LIN {X 0,Y 210.828,Z 695.055,A -85,B 0,C 180,E1 -21900.557,E2 -21900.557} C_VEL
LIN {X 0,Y 214.212,Z 683.602,A -85,B 0,C 180,E1 -21902.499,E2 -21902.499} C_VEL
LIN {X 0,Y 216.871,Z 672.44,A -85,B 0,C 180,E1 -21903.99,E2 -21903.99} C_VEL
LIN {X 0,Y 219.279,Z 660.117,A -85,B 0,C 180,E1 -21905.236,E2 -21905.236} C_VEL
LIN {X 0,Y 220.903,Z 648.24,A -85,B 0,C 180,E1 -21906.129,E2 -21906.129} C_VEL
LIN {X 0,Y 222.158,Z 635.708,A -85,B 0,C 180,E1 -21906.737,E2 -21906.737} C_VEL
LIN {X 0,Y 225.382,Z 570.119,A -85,B 0,C 180,E1 -21908.634,E2 -21908.634} C_VEL
LIN {X 0,Y 224.372,Z 564.639,A -85,B 0,C 180,E1 -21909.068,E2 -21909.068} C_VEL
LIN {X 0,Y 218.505,Z 551.425,A -85,B 0,C 180,E1 -21910.952,E2 -21910.952} C_VEL
LIN {X 0,Y 212.899,Z 540.525,A -85,B 0,C 180,E1 -21912.833,E2 -21912.833} C_VEL
LIN {X 0,Y 207.547,Z 531.361,A -85,B 0,C 180,E1 -21914.735,E2 -21914.735} C_VEL
LIN {X 0,Y 204.869,Z 527.036,A -85,B 0,C 180,E1 -21915.738,E2 -21915.738} C_VEL
LIN {X 0,Y 202.022,Z 522.55,A -85,B 0,C 180,E1 -21916.851,E2 -21916.851} C_VEL
LIN {X 0,Y 199.415,Z 518.27,A -85,B 0,C 180,E1 -21917.962,E2 -21917.962} C_VEL
LIN {X 0,Y 197.926,Z 513.312,A -85,B 0,C 180,E1 -21921.372,E2 -21921.372} C_VEL
LIN {X 0,Y 197,Z 511.784,A -85,B 0,C 180,E1 -21922.664,E2 -21922.664} C_VEL
LIN {X 0,Y 195.61,Z 510.693,A -85,B 0,C 180,E1 -21924.04,E2 -21924.04} C_VEL
LIN {X 0,Y 199.723,Z 529.401,A -85,B 0,C 180,E1 -21929.32,E2 -21929.32} C_VEL
LIN {X 0,Y 199.82,Z 531.676,A -85,B 0,C 180,E1 -21929.92,E2 -21929.92} C_VEL
LIN {X 0,Y 199.088,Z 537.434,A -85,B 0,C 180,E1 -21931.377,E2 -21931.377} C_VEL
LIN {X 0,Y 200.579,Z 559.049,A -85,B 0,C 180,E1 -21932.803,E2 -21932.803} C_VEL
LIN {X 0,Y 201.371,Z 568.64,A -85,B 0,C 180,E1 -21933.438,E2 -21933.438} C_VEL
LIN {X 0,Y 197.17,Z 649.531,A -85,B 0,C 180,E1 -21938.537,E2 -21938.537} C_VEL
LIN {X 0,Y 196.297,Z 664.074,A -85,B 0,C 180,E1 -21939.842,E2 -21939.842} C_VEL
LIN {X 0,Y 195.289,Z 676.673,A -85,B 0,C 180,E1 -21941.374,E2 -21941.374} C_VEL
LIN {X 0,Y 194.349,Z 688.461,A -85,B 0,C 180,E1 -21943.184,E2 -21943.184} C_VEL
LIN {X 0,Y 193.196,Z 700.417,A -85,B 0,C 180,E1 -21945.516,E2 -21945.516} C_VEL
LIN {X 0,Y 192.294,Z 710.299,A -85,B 0,C 180,E1 -21947.868,E2 -21947.868} C_VEL
LIN {X 0,Y 191.618,Z 719.434,A -85,B 0,C 180,E1 -21950.5,E2 -21950.5} C_VEL
LIN {X 0,Y 190.999,Z 728.454,A -85,B 0,C 180,E1 -21953.662,E2 -21953.662} C_VEL
LIN {X 0,Y 190.744,Z 735.772,A -85,B 0,C 180,E1 -21956.831,E2 -21956.831} C_VEL
LIN {X 0,Y 190.589,Z 741.573,A -85,B 0,C 180,E1 -21960,E2 -21960} C_VEL
LIN {X 0,Y 190.77,Z 746.231,A -85,B 0,C 180,E1 -21963.167,E2 -21963.167} C_VEL
LIN {X 0,Y 191.186,Z 749.856,A -85,B 0,C 180,E1 -21966.331,E2 -21966.331} C_VEL
LIN {X 0,Y 192.742,Z 753.216,A -85,B 0,C 180,E1 -21970.504,E2 -21970.504} C_VEL
LIN {X 0,Y 195.223,Z 755.083,A -85,B 0,C 180,E1 -21974.596,E2 -21974.596} C_VEL
LIN {X 0,Y 198.727,Z 755.426,A -85,B 0,C 180,E1 -21978.559,E2 -21978.559} C_VEL
LIN {X 0,Y 200.496,Z 755.13,A -85,B 0,C 180,E1 -21980.073,E2 -21980.073} C_VEL
LIN {X 0,Y 201.902,Z 754.816,A -85,B 0,C 180,E1 -21981.708,E2 -21981.708} C_VEL
LIN {X 0,Y 202.92,Z 754.106,A -85,B 0,C 180,E1 -21984.496,E2 -21984.496} C_VEL
LIN {X 0,Y 204.459,Z 752.722,A -85,B 0,C 180,E1 -21987.21,E2 -21987.21} C_VEL
LIN {X 0,Y 206.611,Z 751.36,A -85,B 0,C 180,E1 -21988.685,E2 -21988.685} C_VEL
LIN {X 0,Y 211.655,Z 748.402,A -85,B 0,C 180,E1 -21990.976,E2 -21990.976} C_VEL
LIN {X 0,Y 217.634,Z 744.305,A -85,B 0,C 180,E1 -21993.297,E2 -21993.297} C_VEL
LIN {X 0,Y 226.261,Z 737.268,A -85,B 0,C 180,E1 -21996.169,E2 -21996.169} C_VEL
LIN {X 0,Y 234.4,Z 729.413,A -85,B 0,C 180,E1 -21998.473,E2 -21998.473} C_VEL
LIN {X 0,Y 241.755,Z 721.254,A -85,B 0,C 180,E1 -22000.296,E2 -22000.296} C_VEL
LIN {X 0,Y 249.501,Z 711.354,A -85,B 0,C 180,E1 -22001.989,E2 -22001.989} C_VEL
LIN {X 0,Y 256.259,Z 701.388,A -85,B 0,C 180,E1 -22003.285,E2 -22003.285} C_VEL
LIN {X 0,Y 257.647,Z 699.121,A -85,B 0,C 180,E1 -22003.543,E2 -22003.543} C_VEL
LIN {X 0,Y 256.765,Z 700.563,A -85,B 0,C 180,E1 -22004.067,E2 -22004.067} C_VEL
LIN {X 0,Y 249.452,Z 711.541,A -85,B 0,C 180,E1 -22005.221,E2 -22005.221} C_VEL
LIN {X 0,Y 241.059,Z 722.516,A -85,B 0,C 180,E1 -22006.791,E2 -22006.791} C_VEL
LIN {X 0,Y 233.324,Z 731.543,A -85,B 0,C 180,E1 -22008.494,E2 -22008.494} C_VEL
LIN {X 0,Y 226.032,Z 739.224,A -85,B 0,C 180,E1 -22010.399,E2 -22010.399} C_VEL
LIN {X 0,Y 217.027,Z 747.683,A -85,B 0,C 180,E1 -22013.193,E2 -22013.193} C_VEL
LIN {X 0,Y 208.803,Z 754.491,A -85,B 0,C 180,E1 -22016.262,E2 -22016.262} C_VEL
LIN {X 0,Y 201.65,Z 759.675,A -85,B 0,C 180,E1 -22019.642,E2 -22019.642} C_VEL
LIN {X 0,Y 197.099,Z 762.649,A -85,B 0,C 180,E1 -22022.381,E2 -22022.381} C_VEL
LIN {X 0,Y 191.959,Z 765.427,A -85,B 0,C 180,E1 -22026.248,E2 -22026.248} C_VEL
LIN {X 0,Y 188.105,Z 766.907,A -85,B 0,C 180,E1 -22030.348,E2 -22030.348} C_VEL
LIN {X 0,Y 185.369,Z 767.073,A -85,B 0,C 180,E1 -22034.607,E2 -22034.607} C_VEL
LIN {X 0,Y 183.999,Z 765.909,A -85,B 0,C 180,E1 -22038.987,E2 -22038.987} C_VEL
LIN {X 0,Y 183.767,Z 765.13,A -85,B 0,C 180,E1 -22040.92,E2 -22040.92} C_VEL
LIN {X 0,Y 183.396,Z 767.379,A -85,B 0,C 180,E1 -22045.106,E2 -22045.106} C_VEL
LIN {X 0,Y 183.43,Z 768.143,A -85,B 0,C 180,E1 -22047.801,E2 -22047.801} C_VEL
LIN {X 0,Y 183.558,Z 768.339,A -85,B 0,C 180,E1 -22049.997,E2 -22049.997} C_VEL
LIN {X 0,Y 183.413,Z 768.131,A -85,B 0,C 180,E1 -22052.193,E2 -22052.193} C_VEL
LIN {X 0,Y 183.327,Z 767.457,A -85,B 0,C 180,E1 -22054.633,E2 -22054.633} C_VEL
LIN {X 0,Y 183.387,Z 765.269,A -85,B 0,C 180,E1 -22058.815,E2 -22058.815} C_VEL
LIN {X 0,Y 184.151,Z 761.471,A -85,B 0,C 180,E1 -22063.234,E2 -22063.234} C_VEL
LIN {X 0,Y 185.381,Z 757.542,A -85,B 0,C 180,E1 -22066.516,E2 -22066.516} C_VEL
LIN {X 0,Y 187.397,Z 751.592,A -85,B 0,C 180,E1 -22070.351,E2 -22070.351} C_VEL
LIN {X 0,Y 190.272,Z 744.3,A -85,B 0,C 180,E1 -22073.969,E2 -22073.969} C_VEL
LIN {X 0,Y 193.247,Z 736.493,A -85,B 0,C 180,E1 -22077.036,E2 -22077.036} C_VEL
LIN {X 0,Y 196.955,Z 727.05,A -85,B 0,C 180,E1 -22079.968,E2 -22079.968} C_VEL
LIN {X 0,Y 200.198,Z 717.757,A -85,B 0,C 180,E1 -22082.301,E2 -22082.301} C_VEL
LIN {X 0,Y 203.605,Z 707.268,A -85,B 0,C 180,E1 -22084.415,E2 -22084.415} C_VEL
LIN {X 0,Y 206.844,Z 696.235,A -85,B 0,C 180,E1 -22086.179,E2 -22086.179} C_VEL
LIN {X 0,Y 209.885,Z 684.296,A -85,B 0,C 180,E1 -22087.666,E2 -22087.666} C_VEL
LIN {X 0,Y 212.604,Z 671.105,A -85,B 0,C 180,E1 -22088.905,E2 -22088.905} C_VEL
LIN {X 0,Y 214.85,Z 656.647,A -85,B 0,C 180,E1 -22089.858,E2 -22089.858} C_VEL
LIN {X 0,Y 216.022,Z 643.586,A -85,B 0,C 180,E1 -22090.436,E2 -22090.436} C_VEL
LIN {X 0,Y 220.134,Z 574.23,A -85,B 0,C 180,E1 -22092.584,E2 -22092.584} C_VEL
LIN {X 0,Y 219.699,Z 569.708,A -85,B 0,C 180,E1 -22092.882,E2 -22092.882} C_VEL
LIN {X 0,Y 214.201,Z 557.072,A -85,B 0,C 180,E1 -22094.776,E2 -22094.776} C_VEL
LIN {X 0,Y 207.641,Z 543.937,A -85,B 0,C 180,E1 -22097.148,E2 -22097.148} C_VEL
LIN {X 0,Y 201.795,Z 533.874,A -85,B 0,C 180,E1 -22099.396,E2 -22099.396} C_VEL
LIN {X 0,Y 199.291,Z 529.804,A -85,B 0,C 180,E1 -22100.417,E2 -22100.417} C_VEL
LIN {X 0,Y 195.906,Z 524.595,A -85,B 0,C 180,E1 -22101.858,E2 -22101.858} C_VEL
LIN {X 0,Y 193.207,Z 520.221,A -85,B 0,C 180,E1 -22103.15,E2 -22103.15} C_VEL
LIN {X 0,Y 191.074,Z 513.748,A -85,B 0,C 180,E1 -22107.771,E2 -22107.771} C_VEL
LIN {X 0,Y 189.183,Z 508.275,A -85,B 0,C 180,E1 -22112.332,E2 -22112.332} C_VEL
LIN {X 0,Y 187.051,Z 502.866,A -85,B 0,C 180,E1 -22117.931,E2 -22117.931} C_VEL
LIN {X 0,Y 185.7,Z 498.97,A -85,B 0,C 180,E1 -22122.944,E2 -22122.944} C_VEL
LIN {X 0,Y 185.933,Z 498.935,A -85,B 0,C 180,E1 -22129.328,E2 -22129.328} C_VEL
LIN {X 0,Y 185.96,Z 498.929,A -85,B 0,C 180,E1 -22133.49,E2 -22133.49} C_VEL
LIN {X 0,Y 186.2,Z 498.901,A -85,B 0,C 180,E1 -22137.837,E2 -22137.837} C_VEL
LIN {X 0,Y 186.4,Z 498.882,A -85,B 0,C 180,E1 -22140,E2 -22140} C_VEL
LIN {X 0,Y 185.916,Z 498.937,A -85,B 0,C 180,E1 -22144.336,E2 -22144.336} C_VEL
LIN {X 0,Y 186,Z 498.925,A -85,B 0,C 180,E1 -22148.693,E2 -22148.693} C_VEL
LIN {X 0,Y 185.725,Z 498.96,A -85,B 0,C 180,E1 -22153.124,E2 -22153.124} C_VEL
LIN {X 0,Y 185.681,Z 498.967,A -85,B 0,C 180,E1 -22157.626,E2 -22157.626} C_VEL
LIN {X 0,Y 185.615,Z 499.116,A -85,B 0,C 180,E1 -22160.792,E2 -22160.792} C_VEL
LIN {X 0,Y 186.948,Z 502.698,A -85,B 0,C 180,E1 -22165.554,E2 -22165.554} C_VEL
LIN {X 0,Y 188.337,Z 506.679,A -85,B 0,C 180,E1 -22169.841,E2 -22169.841} C_VEL
LIN {X 0,Y 189.408,Z 509.491,A -85,B 0,C 180,E1 -22172.55,E2 -22172.55} C_VEL
LIN {X 0,Y 190.819,Z 513.625,A -85,B 0,C 180,E1 -22176.107,E2 -22176.107} C_VEL
LIN {X 0,Y 192.368,Z 518.557,A -85,B 0,C 180,E1 -22179.768,E2 -22179.768} C_VEL
LIN {X 0,Y 195.364,Z 523.112,A -85,B 0,C 180,E1 -22181.125,E2 -22181.125} C_VEL
LIN {X 0,Y 199.994,Z 530.331,A -85,B 0,C 180,E1 -22183.083,E2 -22183.083} C_VEL
LIN {X 0,Y 205.293,Z 539.051,A -85,B 0,C 180,E1 -22185.156,E2 -22185.156} C_VEL
LIN {X 0,Y 209.864,Z 547.445,A -85,B 0,C 180,E1 -22186.84,E2 -22186.84} C_VEL
LIN {X 0,Y 216.245,Z 560.626,A -85,B 0,C 180,E1 -22189.054,E2 -22189.054} C_VEL
LIN {X 0,Y 219.375,Z 568.172,A -85,B 0,C 180,E1 -22190.109,E2 -22190.109} C_VEL
LIN {X 0,Y 219.825,Z 571.346,A -85,B 0,C 180,E1 -22190.342,E2 -22190.342} C_VEL
LIN {X 0,Y 216.388,Z 636.763,A -85,B 0,C 180,E1 -22192.268,E2 -22192.268} C_VEL
LIN {X 0,Y 215.017,Z 649.702,A -85,B 0,C 180,E1 -22192.944,E2 -22192.944} C_VEL
LIN {X 0,Y 213.008,Z 662.945,A -85,B 0,C 180,E1 -22194.009,E2 -22194.009} C_VEL
LIN {X 0,Y 210.795,Z 673.823,A -85,B 0,C 180,E1 -22195.187,E2 -22195.187} C_VEL
LIN {X 0,Y 207.573,Z 686.197,A -85,B 0,C 180,E1 -22196.913,E2 -22196.913} C_VEL
LIN {X 0,Y 204.193,Z 697.188,A -85,B 0,C 180,E1 -22198.92,E2 -22198.92} C_VEL
LIN {X 0,Y 200.881,Z 706.917,A -85,B 0,C 180,E1 -22201.204,E2 -22201.204} C_VEL
LIN {X 0,Y 197.666,Z 715.222,A -85,B 0,C 180,E1 -22203.616,E2 -22203.616} C_VEL
LIN {X 0,Y 194.244,Z 723.284,A -85,B 0,C 180,E1 -22206.55,E2 -22206.55} C_VEL
LIN {X 0,Y 191.401,Z 729.836,A -85,B 0,C 180,E1 -22209.587,E2 -22209.587} C_VEL
LIN {X 0,Y 188.956,Z 735.137,A -85,B 0,C 180,E1 -22212.693,E2 -22212.693} C_VEL
LIN {X 0,Y 186.916,Z 739.358,A -85,B 0,C 180,E1 -22215.857,E2 -22215.857} C_VEL
LIN {X 0,Y 185.491,Z 742.602,A -85,B 0,C 180,E1 -22219.083,E2 -22219.083} C_VEL
LIN {X 0,Y 184.306,Z 745.494,A -85,B 0,C 180,E1 -22223.434,E2 -22223.434} C_VEL
LIN {X 0,Y 183.971,Z 746.394,A -85,B 0,C 180,E1 -22225.621,E2 -22225.621} C_VEL
LIN {X 0,Y 183.613,Z 747.151,A -85,B 0,C 180,E1 -22230.003,E2 -22230.003} C_VEL
LIN {X 0,Y 183.967,Z 746.444,A -85,B 0,C 180,E1 -22234.385,E2 -22234.385} C_VEL
LIN {X 0,Y 184.82,Z 744.322,A -85,B 0,C 180,E1 -22238.752,E2 -22238.752} C_VEL
LIN {X 0,Y 186.363,Z 740.712,A -85,B 0,C 180,E1 -22243.08,E2 -22243.08} C_VEL
LIN {X 0,Y 188.182,Z 736.87,A -85,B 0,C 180,E1 -22246.269,E2 -22246.269} C_VEL
LIN {X 0,Y 190.453,Z 731.988,A -85,B 0,C 180,E1 -22249.4,E2 -22249.4} C_VEL
LIN {X 0,Y 193.666,Z 724.806,A -85,B 0,C 180,E1 -22252.964,E2 -22252.964} C_VEL
LIN {X 0,Y 197.069,Z 717.059,A -85,B 0,C 180,E1 -22255.907,E2 -22255.907} C_VEL
LIN {X 0,Y 200.605,Z 707.966,A -85,B 0,C 180,E1 -22258.652,E2 -22258.652} C_VEL
LIN {X 0,Y 204.077,Z 697.743,A -85,B 0,C 180,E1 -22261.105,E2 -22261.105} C_VEL
LIN {X 0,Y 207.488,Z 686.919,A -85,B 0,C 180,E1 -22263.108,E2 -22263.108} C_VEL
LIN {X 0,Y 210.663,Z 674.74,A -85,B 0,C 180,E1 -22264.844,E2 -22264.844} C_VEL
LIN {X 0,Y 213.349,Z 661.864,A -85,B 0,C 180,E1 -22266.223,E2 -22266.223} C_VEL
LIN {X 0,Y 215.228,Z 648.999,A -85,B 0,C 180,E1 -22267.24,E2 -22267.24} C_VEL
LIN {X 0,Y 216.629,Z 635.409,A -85,B 0,C 180,E1 -22267.91,E2 -22267.91} C_VEL
LIN {X 0,Y 219.891,Z 570.921,A -85,B 0,C 180,E1 -22269.819,E2 -22269.819} C_VEL
LIN {X 0,Y 219.169,Z 567.413,A -85,B 0,C 180,E1 -22270.129,E2 -22270.129} C_VEL
LIN {X 0,Y 213.489,Z 554.633,A -85,B 0,C 180,E1 -22272.056,E2 -22272.056} C_VEL
LIN {X 0,Y 207.921,Z 543.686,A -85,B 0,C 180,E1 -22274.045,E2 -22274.045} C_VEL
LIN {X 0,Y 201.735,Z 533.018,A -85,B 0,C 180,E1 -22276.407,E2 -22276.407} C_VEL
LIN {X 0,Y 195.52,Z 523.284,A -85,B 0,C 180,E1 -22279.005,E2 -22279.005} C_VEL
LIN {X 0,Y 192.488,Z 518.803,A -85,B 0,C 180,E1 -22280.378,E2 -22280.378} C_VEL
LIN {X 0,Y 192.114,Z 517.754,A -85,B 0,C 180,E1 -22280.967,E2 -22280.967} C_VEL
LIN {X 0,Y 191.064,Z 515.766,A -85,B 0,C 180,E1 -22282.632,E2 -22282.632} C_VEL
LIN {X 0,Y 189.174,Z 514.41,A -85,B 0,C 180,E1 -22284.502,E2 -22284.502} C_VEL
LIN {X 0,Y 192.821,Z 531.138,A -85,B 0,C 180,E1 -22289.317,E2 -22289.317} C_VEL
LIN {X 0,Y 192.104,Z 538.019,A -85,B 0,C 180,E1 -22291.064,E2 -22291.064} C_VEL
LIN {X 0,Y 193.569,Z 559.593,A -85,B 0,C 180,E1 -22292.556,E2 -22292.556} C_VEL
LIN {X 0,Y 194.309,Z 568.869,A -85,B 0,C 180,E1 -22293.193,E2 -22293.193} C_VEL
LIN {X 0,Y 190.046,Z 649.637,A -85,B 0,C 180,E1 -22298.51,E2 -22298.51} C_VEL
LIN {X 0,Y 189.174,Z 664.364,A -85,B 0,C 180,E1 -22299.9,E2 -22299.9} C_VEL
LIN {X 0,Y 188.01,Z 678.656,A -85,B 0,C 180,E1 -22301.755,E2 -22301.755} C_VEL
LIN {X 0,Y 186.909,Z 691.344,A -85,B 0,C 180,E1 -22303.9,E2 -22303.9} C_VEL
LIN {X 0,Y 185.841,Z 702.867,A -85,B 0,C 180,E1 -22306.328,E2 -22306.328} C_VEL
LIN {X 0,Y 185.015,Z 713.367,A -85,B 0,C 180,E1 -22309.051,E2 -22309.051} C_VEL
LIN {X 0,Y 184.336,Z 722.232,A -85,B 0,C 180,E1 -22311.835,E2 -22311.835} C_VEL
LIN {X 0,Y 183.844,Z 730.576,A -85,B 0,C 180,E1 -22315.084,E2 -22315.084} C_VEL
LIN {X 0,Y 183.65,Z 737.43,A -85,B 0,C 180,E1 -22318.355,E2 -22318.355} C_VEL
LIN {X 0,Y 183.659,Z 743.84,A -85,B 0,C 180,E1 -22322.193,E2 -22322.193} C_VEL
LIN {X 0,Y 183.982,Z 748.054,A -85,B 0,C 180,E1 -22325.48,E2 -22325.48} C_VEL
LIN {X 0,Y 184.801,Z 751.311,A -85,B 0,C 180,E1 -22328.75,E2 -22328.75} C_VEL
LIN {X 0,Y 185.773,Z 753.008,A -85,B 0,C 180,E1 -22330.903,E2 -22330.903} C_VEL
LIN {X 0,Y 188.382,Z 755.215,A -85,B 0,C 180,E1 -22335.138,E2 -22335.138} C_VEL
LIN {X 0,Y 192.038,Z 756.004,A -85,B 0,C 180,E1 -22339.23,E2 -22339.23} C_VEL
LIN {X 0,Y 196.892,Z 755.347,A -85,B 0,C 180,E1 -22343.119,E2 -22343.119} C_VEL
LIN {X 0,Y 202.881,Z 753.185,A -85,B 0,C 180,E1 -22346.765,E2 -22346.765} C_VEL
LIN {X 0,Y 206.611,Z 751.36,A -85,B 0,C 180,E1 -22348.685,E2 -22348.685} C_VEL
LIN {X 0,Y 208.987,Z 749.912,A -85,B 0,C 180,E1 -22350.123,E2 -22350.123} C_VEL
LIN {X 0,Y 214.267,Z 745.594,A -85,B 0,C 180,E1 -22354.582,E2 -22354.582} C_VEL
LIN {X 0,Y 216.855,Z 743.551,A -85,B 0,C 180,E1 -22355.871,E2 -22355.871} C_VEL
LIN {X 0,Y 217.926,Z 742.732,A -85,B 0,C 180,E1 -22356.246,E2 -22356.246} C_VEL
LIN {X 0,Y 225.662,Z 736.578,A -85,B 0,C 180,E1 -22358.526,E2 -22358.526} C_VEL
LIN {X 0,Y 234.459,Z 728.429,A -85,B 0,C 180,E1 -22360.729,E2 -22360.729} C_VEL
LIN {X 0,Y 242.237,Z 720.047,A -85,B 0,C 180,E1 -22362.419,E2 -22362.419} C_VEL
LIN {X 0,Y 246.299,Z 715.233,A -85,B 0,C 180,E1 -22363.222,E2 -22363.222} C_VEL
LIN {X 0,Y 247.031,Z 714.366,A -85,B 0,C 180,E1 -22363.811,E2 -22363.811} C_VEL
LIN {X 0,Y 237.76,Z 725.357,A -85,B 0,C 180,E1 -22365.428,E2 -22365.428} C_VEL
LIN {X 0,Y 228.369,Z 735.123,A -85,B 0,C 180,E1 -22367.384,E2 -22367.384} C_VEL
LIN {X 0,Y 219.714,Z 743.094,A -85,B 0,C 180,E1 -22369.626,E2 -22369.626} C_VEL
LIN {X 0,Y 211.56,Z 749.776,A -85,B 0,C 180,E1 -22372.077,E2 -22372.077} C_VEL
LIN {X 0,Y 205.079,Z 754.54,A -85,B 0,C 180,E1 -22374.365,E2 -22374.365} C_VEL
LIN {X 0,Y 197.388,Z 759.54,A -85,B 0,C 180,E1 -22377.716,E2 -22377.716} C_VEL
LIN {X 0,Y 190.848,Z 763.176,A -85,B 0,C 180,E1 -22381.395,E2 -22381.395} C_VEL
LIN {X 0,Y 185.175,Z 765.594,A -85,B 0,C 180,E1 -22385.627,E2 -22385.627} C_VEL
LIN {X 0,Y 181.412,Z 766.552,A -85,B 0,C 180,E1 -22389.591,E2 -22389.591} C_VEL
LIN {X 0,Y 178.534,Z 766.312,A -85,B 0,C 180,E1 -22394.002,E2 -22394.002} C_VEL
LIN {X 0,Y 177.08,Z 764.778,A -85,B 0,C 180,E1 -22398.551,E2 -22398.551} C_VEL
LIN {X 0,Y 176.915,Z 764.245,A -85,B 0,C 180,E1 -22399.844,E2 -22399.844} C_VEL
LIN {X 0,Y 176.377,Z 766.218,A -85,B 0,C 180,E1 -22403.132,E2 -22403.132} C_VEL
LIN {X 0,Y 176.347,Z 767.734,A -85,B 0,C 180,E1 -22407.713,E2 -22407.713} C_VEL
LIN {X 0,Y 176.491,Z 767.931,A -85,B 0,C 180,E1 -22409.997,E2 -22409.997} C_VEL
LIN {X 0,Y 176.328,Z 767.721,A -85,B 0,C 180,E1 -22412.281,E2 -22412.281} C_VEL
LIN {X 0,Y 176.26,Z 767.139,A -85,B 0,C 180,E1 -22414.571,E2 -22414.571} C_VEL
LIN {X 0,Y 176.319,Z 764.855,A -85,B 0,C 180,E1 -22419.171,E2 -22419.171} C_VEL
LIN {X 0,Y 177.185,Z 761.055,A -85,B 0,C 180,E1 -22423.765,E2 -22423.765} C_VEL
LIN {X 0,Y 178.502,Z 757.122,A -85,B 0,C 180,E1 -22427.172,E2 -22427.172} C_VEL
LIN {X 0,Y 180.48,Z 751.68,A -85,B 0,C 180,E1 -22430.841,E2 -22430.841} C_VEL
LIN {X 0,Y 183.261,Z 745.018,A -85,B 0,C 180,E1 -22434.343,E2 -22434.343} C_VEL
LIN {X 0,Y 186.33,Z 737.443,A -85,B 0,C 180,E1 -22437.516,E2 -22437.516} C_VEL
LIN {X 0,Y 190.104,Z 728.28,A -85,B 0,C 180,E1 -22440.549,E2 -22440.549} C_VEL
LIN {X 0,Y 194.041,Z 717.72,A -85,B 0,C 180,E1 -22443.328,E2 -22443.328} C_VEL
LIN {X 0,Y 197.756,Z 706.772,A -85,B 0,C 180,E1 -22445.584,E2 -22445.584} C_VEL
LIN {X 0,Y 201.135,Z 695.701,A -85,B 0,C 180,E1 -22447.377,E2 -22447.377} C_VEL
LIN {X 0,Y 204.284,Z 683.703,A -85,B 0,C 180,E1 -22448.888,E2 -22448.888} C_VEL
LIN {X 0,Y 207.118,Z 670.419,A -85,B 0,C 180,E1 -22450.141,E2 -22450.141} C_VEL
LIN {X 0,Y 209.312,Z 656.694,A -85,B 0,C 180,E1 -22451.056,E2 -22451.056} C_VEL
LIN {X 0,Y 210.642,Z 642.34,A -85,B 0,C 180,E1 -22451.694,E2 -22451.694} C_VEL
LIN {X 0,Y 214.737,Z 574.401,A -85,B 0,C 180,E1 -22453.84,E2 -22453.84} C_VEL
LIN {X 0,Y 214.275,Z 571.884,A -85,B 0,C 180,E1 -22454.069,E2 -22454.069} C_VEL
LIN {X 0,Y 208.862,Z 559.406,A -85,B 0,C 180,E1 -22456.052,E2 -22456.052} C_VEL
LIN {X 0,Y 203.18,Z 548.01,A -85,B 0,C 180,E1 -22458.234,E2 -22458.234} C_VEL
LIN {X 0,Y 197.7,Z 538.379,A -85,B 0,C 180,E1 -22460.47,E2 -22460.47} C_VEL
LIN {X 0,Y 192.866,Z 530.492,A -85,B 0,C 180,E1 -22462.607,E2 -22462.607} C_VEL
LIN {X 0,Y 189.054,Z 524.849,A -85,B 0,C 180,E1 -22464.408,E2 -22464.408} C_VEL
LIN {X 0,Y 186.008,Z 520.154,A -85,B 0,C 180,E1 -22466.014,E2 -22466.014} C_VEL
LIN {X 0,Y 184.229,Z 514.815,A -85,B 0,C 180,E1 -22470.269,E2 -22470.269} C_VEL
LIN {X 0,Y 183.06,Z 511.65,A -85,B 0,C 180,E1 -22473.211,E2 -22473.211} C_VEL
LIN {X 0,Y 181.622,Z 507.861,A -85,B 0,C 180,E1 -22477.235,E2 -22477.235} C_VEL
LIN {X 0,Y 180.249,Z 504.26,A -85,B 0,C 180,E1 -22481.825,E2 -22481.825} C_VEL
LIN {X 0,Y 179.688,Z 502.737,A -85,B 0,C 180,E1 -22484.111,E2 -22484.111} C_VEL
LIN {X 0,Y 178.887,Z 499.814,A -85,B 0,C 180,E1 -22489.646,E2 -22489.646} C_VEL
LIN {X 0,Y 178.925,Z 499.806,A -85,B 0,C 180,E1 -22493.233,E2 -22493.233} C_VEL
LIN {X 0,Y 179.146,Z 499.78,A -85,B 0,C 180,E1 -22497.752,E2 -22497.752} C_VEL
LIN {X 0,Y 179.363,Z 499.758,A -85,B 0,C 180,E1 -22500,E2 -22500} C_VEL
LIN {X 0,Y 178.864,Z 499.816,A -85,B 0,C 180,E1 -22504.508,E2 -22504.508} C_VEL
LIN {X 0,Y 178.929,Z 499.806,A -85,B 0,C 180,E1 -22509.04,E2 -22509.04} C_VEL
LIN {X 0,Y 178.66,Z 499.954,A -85,B 0,C 180,E1 -22514.233,E2 -22514.233} C_VEL
LIN {X 0,Y 179.953,Z 503.316,A -85,B 0,C 180,E1 -22520.579,E2 -22520.579} C_VEL
LIN {X 0,Y 181.157,Z 506.732,A -85,B 0,C 180,E1 -22525.262,E2 -22525.262} C_VEL
LIN {X 0,Y 182.245,Z 509.852,A -85,B 0,C 180,E1 -22528.819,E2 -22528.819} C_VEL
LIN {X 0,Y 183.61,Z 513.695,A -85,B 0,C 180,E1 -22532.645,E2 -22532.645} C_VEL
LIN {X 0,Y 185.303,Z 518.732,A -85,B 0,C 180,E1 -22536.902,E2 -22536.902} C_VEL
LIN {X 0,Y 188.358,Z 523.244,A -85,B 0,C 180,E1 -22538.473,E2 -22538.473} C_VEL
LIN {X 0,Y 190.015,Z 525.741,A -85,B 0,C 180,E1 -22539.283,E2 -22539.283} C_VEL
LIN {X 0,Y 193.208,Z 530.477,A -85,B 0,C 180,E1 -22540.761,E2 -22540.761} C_VEL
LIN {X 0,Y 199.397,Z 540.507,A -85,B 0,C 180,E1 -22543.417,E2 -22543.417} C_VEL
LIN {X 0,Y 205.095,Z 550.84,A -85,B 0,C 180,E1 -22545.666,E2 -22545.666} C_VEL
LIN {X 0,Y 211.384,Z 564.046,A -85,B 0,C 180,E1 -22547.984,E2 -22547.984} C_VEL
LIN {X 0,Y 214.297,Z 571.246,A -85,B 0,C 180,E1 -22549.03,E2 -22549.03} C_VEL
LIN {X 0,Y 214.507,Z 572.611,A -85,B 0,C 180,E1 -22549.139,E2 -22549.139} C_VEL
LIN {X 0,Y 210.819,Z 637.812,A -85,B 0,C 180,E1 -22551.087,E2 -22551.087} C_VEL
LIN {X 0,Y 209.428,Z 650.464,A -85,B 0,C 180,E1 -22551.78,E2 -22551.78} C_VEL
LIN {X 0,Y 207.331,Z 663.577,A -85,B 0,C 180,E1 -22552.861,E2 -22552.861} C_VEL
LIN {X 0,Y 205.045,Z 674.378,A -85,B 0,C 180,E1 -22554.062,E2 -22554.062} C_VEL
LIN {X 0,Y 202.092,Z 685.291,A -85,B 0,C 180,E1 -22555.593,E2 -22555.593} C_VEL
LIN {X 0,Y 198.536,Z 696.55,A -85,B 0,C 180,E1 -22557.632,E2 -22557.632} C_VEL
LIN {X 0,Y 195.268,Z 705.708,A -85,B 0,C 180,E1 -22559.746,E2 -22559.746} C_VEL
LIN {X 0,Y 192.022,Z 714.159,A -85,B 0,C 180,E1 -22562.186,E2 -22562.186} C_VEL
LIN {X 0,Y 188.377,Z 722.5,A -85,B 0,C 180,E1 -22565.187,E2 -22565.187} C_VEL
LIN {X 0,Y 185.295,Z 729.27,A -85,B 0,C 180,E1 -22568.3,E2 -22568.3} C_VEL
LIN {X 0,Y 182.203,Z 735.552,A -85,B 0,C 180,E1 -22572.03,E2 -22572.03} C_VEL
LIN {X 0,Y 180.064,Z 739.769,A -85,B 0,C 180,E1 -22575.307,E2 -22575.307} C_VEL
LIN {X 0,Y 178.528,Z 743.012,A -85,B 0,C 180,E1 -22578.651,E2 -22578.651} C_VEL
LIN {X 0,Y 177.273,Z 745.903,A -85,B 0,C 180,E1 -22583.172,E2 -22583.172} C_VEL
LIN {X 0,Y 176.639,Z 747.357,A -85,B 0,C 180,E1 -22587.723,E2 -22587.723} C_VEL
LIN {X 0,Y 176.638,Z 747.387,A -85,B 0,C 180,E1 -22592.283,E2 -22592.283} C_VEL
LIN {X 0,Y 177.273,Z 745.971,A -85,B 0,C 180,E1 -22596.834,E2 -22596.834} C_VEL
LIN {X 0,Y 178.532,Z 743.121,A -85,B 0,C 180,E1 -22601.354,E2 -22601.354} C_VEL
LIN {X 0,Y 180.063,Z 739.926,A -85,B 0,C 180,E1 -22604.699,E2 -22604.699} C_VEL
LIN {X 0,Y 182.138,Z 735.761,A -85,B 0,C 180,E1 -22607.983,E2 -22607.983} C_VEL
LIN {X 0,Y 184.697,Z 730.514,A -85,B 0,C 180,E1 -22611.195,E2 -22611.195} C_VEL
LIN {X 0,Y 188.278,Z 722.816,A -85,B 0,C 180,E1 -22614.833,E2 -22614.833} C_VEL
LIN {X 0,Y 191.964,Z 714.563,A -85,B 0,C 180,E1 -22617.829,E2 -22617.829} C_VEL
LIN {X 0,Y 195.238,Z 706.192,A -85,B 0,C 180,E1 -22620.265,E2 -22620.265} C_VEL
LIN {X 0,Y 198.786,Z 695.992,A -85,B 0,C 180,E1 -22622.629,E2 -22622.629} C_VEL
LIN {X 0,Y 202.446,Z 684.597,A -85,B 0,C 180,E1 -22624.646,E2 -22624.646} C_VEL
LIN {X 0,Y 205.286,Z 673.531,A -85,B 0,C 180,E1 -22626.199,E2 -22626.199} C_VEL
LIN {X 0,Y 207.917,Z 661.351,A -85,B 0,C 180,E1 -22627.479,E2 -22627.479} C_VEL
LIN {X 0,Y 209.77,Z 648.969,A -85,B 0,C 180,E1 -22628.458,E2 -22628.458} C_VEL
LIN {X 0,Y 211.214,Z 635.111,A -85,B 0,C 180,E1 -22629.139,E2 -22629.139} C_VEL
LIN {X 0,Y 214.56,Z 572.068,A -85,B 0,C 180,E1 -22631.034,E2 -22631.034} C_VEL
LIN {X 0,Y 213.368,Z 568.595,A -85,B 0,C 180,E1 -22631.479,E2 -22631.479} C_VEL
LIN {X 0,Y 207.976,Z 556.519,A -85,B 0,C 180,E1 -22633.432,E2 -22633.432} C_VEL
LIN {X 0,Y 202.314,Z 545.576,A -85,B 0,C 180,E1 -22635.597,E2 -22635.597} C_VEL
LIN {X 0,Y 197.016,Z 536.568,A -85,B 0,C 180,E1 -22637.762,E2 -22637.762} C_VEL
LIN {X 0,Y 191.944,Z 528.466,A -85,B 0,C 180,E1 -22640.022,E2 -22640.022} C_VEL
LIN {X 0,Y 188.295,Z 523.137,A -85,B 0,C 180,E1 -22641.773,E2 -22641.773} C_VEL
LIN {X 0,Y 184.64,Z 519.623,A -85,B 0,C 180,E1 -22643.557,E2 -22643.557} C_VEL
LIN {X 0,Y 182.997,Z 518.35,A -85,B 0,C 180,E1 -22644.5,E2 -22644.5} C_VEL
LIN {X 0,Y 182.722,Z 518.052,A -85,B 0,C 180,E1 -22644.987,E2 -22644.987} C_VEL
LIN {X 0,Y 185.806,Z 532.74,A -85,B 0,C 180,E1 -22649.294,E2 -22649.294} C_VEL
LIN {X 0,Y 185.11,Z 538.389,A -85,B 0,C 180,E1 -22650.737,E2 -22650.737} C_VEL
LIN {X 0,Y 186.607,Z 560.883,A -85,B 0,C 180,E1 -22652.344,E2 -22652.344} C_VEL
LIN {X 0,Y 187.277,Z 569.198,A -85,B 0,C 180,E1 -22652.937,E2 -22652.937} C_VEL
LIN {X 0,Y 183,Z 648.605,A -85,B 0,C 180,E1 -22658.454,E2 -22658.454} C_VEL
LIN {X 0,Y 182.151,Z 663.033,A -85,B 0,C 180,E1 -22659.828,E2 -22659.828} C_VEL
LIN {X 0,Y 181.22,Z 674.898,A -85,B 0,C 180,E1 -22661.34,E2 -22661.34} C_VEL
LIN {X 0,Y 180.089,Z 688.512,A -85,B 0,C 180,E1 -22663.564,E2 -22663.564} C_VEL
LIN {X 0,Y 178.935,Z 700.569,A -85,B 0,C 180,E1 -22666.079,E2 -22666.079} C_VEL
LIN {X 0,Y 178.127,Z 710.464,A -85,B 0,C 180,E1 -22668.622,E2 -22668.622} C_VEL
LIN {X 0,Y 177.445,Z 719.59,A -85,B 0,C 180,E1 -22671.459,E2 -22671.459} C_VEL
LIN {X 0,Y 176.911,Z 728.636,A -85,B 0,C 180,E1 -22674.891,E2 -22674.891} C_VEL
LIN {X 0,Y 176.68,Z 735.94,A -85,B 0,C 180,E1 -22678.29,E2 -22678.29} C_VEL
LIN {X 0,Y 176.663,Z 742.652,A -85,B 0,C 180,E1 -22682.28,E2 -22682.28} C_VEL
LIN {X 0,Y 176.968,Z 747.194,A -85,B 0,C 180,E1 -22685.698,E2 -22685.698} C_VEL
LIN {X 0,Y 177.821,Z 750.753,A -85,B 0,C 180,E1 -22689.096,E2 -22689.096} C_VEL
LIN {X 0,Y 180.023,Z 754.121,A -85,B 0,C 180,E1 -22693.546,E2 -22693.546} C_VEL
LIN {X 0,Y 183.309,Z 756.044,A -85,B 0,C 180,E1 -22697.861,E2 -22697.861} C_VEL
LIN {X 0,Y 185.382,Z 756.465,A -85,B 0,C 180,E1 -22699.95,E2 -22699.95} C_VEL
LIN {X 0,Y 190.449,Z 756.219,A -85,B 0,C 180,E1 -22703.949,E2 -22703.949} C_VEL
LIN {X 0,Y 196.686,Z 754.575,A -85,B 0,C 180,E1 -22707.679,E2 -22707.679} C_VEL
LIN {X 0,Y 203.882,Z 751.474,A -85,B 0,C 180,E1 -22711.135,E2 -22711.135} C_VEL
LIN {X 0,Y 212.024,Z 746.782,A -85,B 0,C 180,E1 -22714.298,E2 -22714.298} C_VEL
LIN {X 0,Y 217.926,Z 742.732,A -85,B 0,C 180,E1 -22716.246,E2 -22716.246} C_VEL
LIN {X 0,Y 220.973,Z 740.356,A -85,B 0,C 180,E1 -22717.418,E2 -22717.418} C_VEL
LIN {X 0,Y 228.483,Z 733.693,A -85,B 0,C 180,E1 -22721.173,E2 -22721.173} C_VEL
LIN {X 0,Y 231.577,Z 730.826,A -85,B 0,C 180,E1 -22722.186,E2 -22722.186} C_VEL
LIN {X 0,Y 232.755,Z 729.734,A -85,B 0,C 180,E1 -22722.459,E2 -22722.459} C_VEL
LIN {X 0,Y 236.253,Z 726.426,A -85,B 0,C 180,E1 -22723.172,E2 -22723.172} C_VEL
LIN {X 0,Y 236.701,Z 726.012,A -85,B 0,C 180,E1 -22723.655,E2 -22723.655} C_VEL
LIN {X 0,Y 227.251,Z 735.122,A -85,B 0,C 180,E1 -22725.424,E2 -22725.424} C_VEL
LIN {X 0,Y 218.311,Z 742.747,A -85,B 0,C 180,E1 -22727.462,E2 -22727.462} C_VEL
LIN {X 0,Y 208.514,Z 750.153,A -85,B 0,C 180,E1 -22730.176,E2 -22730.176} C_VEL
LIN {X 0,Y 201.634,Z 754.672,A -85,B 0,C 180,E1 -22732.41,E2 -22732.41} C_VEL
LIN {X 0,Y 193.35,Z 759.471,A -85,B 0,C 180,E1 -22735.706,E2 -22735.706} C_VEL
LIN {X 0,Y 187.893,Z 762.142,A -85,B 0,C 180,E1 -22738.419,E2 -22738.419} C_VEL
LIN {X 0,Y 181.742,Z 764.636,A -85,B 0,C 180,E1 -22742.349,E2 -22742.349} C_VEL
LIN {X 0,Y 176.737,Z 765.908,A -85,B 0,C 180,E1 -22746.565,E2 -22746.565} C_VEL
LIN {X 0,Y 173.103,Z 765.927,A -85,B 0,C 180,E1 -22751.043,E2 -22751.043} C_VEL
LIN {X 0,Y 170.795,Z 764.655,A -85,B 0,C 180,E1 -22755.703,E2 -22755.703} C_VEL
LIN {X 0,Y 170.082,Z 763.284,A -85,B 0,C 180,E1 -22758.678,E2 -22758.678} C_VEL
LIN {X 0,Y 169.325,Z 765.808,A -85,B 0,C 180,E1 -22762.844,E2 -22762.844} C_VEL
LIN {X 0,Y 169.215,Z 766.812,A -85,B 0,C 180,E1 -22765.405,E2 -22765.405} C_VEL
LIN {X 0,Y 169.403,Z 767.522,A -85,B 0,C 180,E1 -22769.997,E2 -22769.997} C_VEL
LIN {X 0,Y 169.174,Z 766.851,A -85,B 0,C 180,E1 -22774.417,E2 -22774.417} C_VEL
LIN {X 0,Y 169.132,Z 765.77,A -85,B 0,C 180,E1 -22777.158,E2 -22777.158} C_VEL
LIN {X 0,Y 169.639,Z 762.736,A -85,B 0,C 180,E1 -22781.952,E2 -22781.952} C_VEL
LIN {X 0,Y 171.155,Z 758.146,A -85,B 0,C 180,E1 -22786.701,E2 -22786.701} C_VEL
LIN {X 0,Y 172.834,Z 753.531,A -85,B 0,C 180,E1 -22790.217,E2 -22790.217} C_VEL
LIN {X 0,Y 175.779,Z 746.834,A -85,B 0,C 180,E1 -22794.19,E2 -22794.19} C_VEL
LIN {X 0,Y 179.415,Z 738.393,A -85,B 0,C 180,E1 -22798.035,E2 -22798.035} C_VEL
LIN {X 0,Y 183.282,Z 729.492,A -85,B 0,C 180,E1 -22801.172,E2 -22801.172} C_VEL
LIN {X 0,Y 187.593,Z 718.617,A -85,B 0,C 180,E1 -22804.188,E2 -22804.188} C_VEL
LIN {X 0,Y 191.57,Z 707.522,A -85,B 0,C 180,E1 -22806.591,E2 -22806.591} C_VEL
LIN {X 0,Y 195.537,Z 695.17,A -85,B 0,C 180,E1 -22808.641,E2 -22808.641} C_VEL
LIN {X 0,Y 198.798,Z 683.113,A -85,B 0,C 180,E1 -22810.175,E2 -22810.175} C_VEL
LIN {X 0,Y 201.724,Z 669.735,A -85,B 0,C 180,E1 -22811.445,E2 -22811.445} C_VEL
LIN {X 0,Y 203.977,Z 655.838,A -85,B 0,C 180,E1 -22812.374,E2 -22812.374} C_VEL
LIN {X 0,Y 205.25,Z 642.568,A -85,B 0,C 180,E1 -22812.966,E2 -22812.966} C_VEL
LIN {X 0,Y 209.486,Z 575.472,A -85,B 0,C 180,E1 -22815.11,E2 -22815.11} C_VEL
LIN {X 0,Y 204.513,Z 563.696,A -85,B 0,C 180,E1 -22817.042,E2 -22817.042} C_VEL
LIN {X 0,Y 199.116,Z 552.696,A -85,B 0,C 180,E1 -22819.234,E2 -22819.234} C_VEL
LIN {X 0,Y 193.471,Z 542.476,A -85,B 0,C 180,E1 -22821.688,E2 -22821.688} C_VEL
LIN {X 0,Y 188.945,Z 535.171,A -85,B 0,C 180,E1 -22823.809,E2 -22823.809} C_VEL
LIN {X 0,Y 185.744,Z 530.224,A -85,B 0,C 180,E1 -22825.42,E2 -22825.42} C_VEL
LIN {X 0,Y 182.221,Z 525.062,A -85,B 0,C 180,E1 -22827.319,E2 -22827.319} C_VEL
LIN {X 0,Y 178.715,Z 520.067,A -85,B 0,C 180,E1 -22829.402,E2 -22829.402} C_VEL
LIN {X 0,Y 177.51,Z 516.172,A -85,B 0,C 180,E1 -22832.915,E2 -22832.915} C_VEL
LIN {X 0,Y 176.221,Z 512.827,A -85,B 0,C 180,E1 -22836.523,E2 -22836.523} C_VEL
LIN {X 0,Y 174.808,Z 509.13,A -85,B 0,C 180,E1 -22841.239,E2 -22841.239} C_VEL
LIN {X 0,Y 174.246,Z 507.515,A -85,B 0,C 180,E1 -22843.601,E2 -22843.601} C_VEL
LIN {X 0,Y 173.395,Z 504.903,A -85,B 0,C 180,E1 -22848.308,E2 -22848.308} C_VEL
LIN {X 0,Y 173.121,Z 503.848,A -85,B 0,C 180,E1 -22850.655,E2 -22850.655} C_VEL
LIN {X 0,Y 172.409,Z 502.061,A -85,B 0,C 180,E1 -22857.664,E2 -22857.664} C_VEL
LIN {X 0,Y 172.532,Z 501.647,A -85,B 0,C 180,E1 -22860,E2 -22860} C_VEL
LIN {X 0,Y 172.296,Z 502.365,A -85,B 0,C 180,E1 -22867.029,E2 -22867.029} C_VEL
LIN {X 0,Y 172.702,Z 503.568,A -85,B 0,C 180,E1 -22871.74,E2 -22871.74} C_VEL
LIN {X 0,Y 173.113,Z 504.362,A -85,B 0,C 180,E1 -22874.099,E2 -22874.099} C_VEL
LIN {X 0,Y 173.853,Z 506.783,A -85,B 0,C 180,E1 -22878.869,E2 -22878.869} C_VEL
LIN {X 0,Y 174.579,Z 508.835,A -85,B 0,C 180,E1 -22882.204,E2 -22882.204} C_VEL
LIN {X 0,Y 176.094,Z 512.722,A -85,B 0,C 180,E1 -22887.368,E2 -22887.368} C_VEL
LIN {X 0,Y 177.648,Z 517.415,A -85,B 0,C 180,E1 -22892.282,E2 -22892.282} C_VEL
LIN {X 0,Y 178.169,Z 518.85,A -85,B 0,C 180,E1 -22893.521,E2 -22893.521} C_VEL
LIN {X 0,Y 181.75,Z 523.817,A -85,B 0,C 180,E1 -22895.632,E2 -22895.632} C_VEL
LIN {X 0,Y 186.602,Z 530.859,A -85,B 0,C 180,E1 -22898.221,E2 -22898.221} C_VEL
LIN {X 0,Y 190.301,Z 536.688,A -85,B 0,C 180,E1 -22900.036,E2 -22900.036} C_VEL
LIN {X 0,Y 195.739,Z 545.66,A -85,B 0,C 180,E1 -22902.484,E2 -22902.484} C_VEL
LIN {X 0,Y 201.034,Z 555.489,A -85,B 0,C 180,E1 -22904.687,E2 -22904.687} C_VEL
LIN {X 0,Y 207.138,Z 568.658,A -85,B 0,C 180,E1 -22907.066,E2 -22907.066} C_VEL
LIN {X 0,Y 209.165,Z 573.586,A -85,B 0,C 180,E1 -22907.829,E2 -22907.829} C_VEL
LIN {X 0,Y 205.491,Z 637.677,A -85,B 0,C 180,E1 -22909.797,E2 -22909.797} C_VEL
LIN {X 0,Y 203.929,Z 651.225,A -85,B 0,C 180,E1 -22910.553,E2 -22910.553} C_VEL
LIN {X 0,Y 201.743,Z 664.208,A -85,B 0,C 180,E1 -22911.649,E2 -22911.649} C_VEL
LIN {X 0,Y 198.921,Z 676.693,A -85,B 0,C 180,E1 -22913.089,E2 -22913.089} C_VEL
LIN {X 0,Y 195.469,Z 688.524,A -85,B 0,C 180,E1 -22914.885,E2 -22914.885} C_VEL
LIN {X 0,Y 191.798,Z 699.172,A -85,B 0,C 180,E1 -22916.975,E2 -22916.975} C_VEL
LIN {X 0,Y 188.322,Z 708.515,A -85,B 0,C 180,E1 -22919.333,E2 -22919.333} C_VEL
LIN {X 0,Y 184.465,Z 717.544,A -85,B 0,C 180,E1 -22922.182,E2 -22922.182} C_VEL
LIN {X 0,Y 180.779,Z 725.338,A -85,B 0,C 180,E1 -22925.3,E2 -22925.3} C_VEL
LIN {X 0,Y 177.227,Z 732.583,A -85,B 0,C 180,E1 -22929.094,E2 -22929.094} C_VEL
LIN {X 0,Y 174.657,Z 737.509,A -85,B 0,C 180,E1 -22932.438,E2 -22932.438} C_VEL
LIN {X 0,Y 172.064,Z 742.432,A -85,B 0,C 180,E1 -22937.021,E2 -22937.021} C_VEL
LIN {X 0,Y 170.519,Z 745.666,A -85,B 0,C 180,E1 -22941.562,E2 -22941.562} C_VEL
LIN {X 0,Y 169.845,Z 747.213,A -85,B 0,C 180,E1 -22945.256,E2 -22945.256} C_VEL
LIN {X 0,Y 169.488,Z 747.966,A -85,B 0,C 180,E1 -22950.003,E2 -22950.003} C_VEL
LIN {X 0,Y 169.841,Z 747.261,A -85,B 0,C 180,E1 -22954.75,E2 -22954.75} C_VEL
LIN {X 0,Y 170.81,Z 745.139,A -85,B 0,C 180,E1 -22959.476,E2 -22959.476} C_VEL
LIN {X 0,Y 172.597,Z 741.53,A -85,B 0,C 180,E1 -22964.144,E2 -22964.144} C_VEL
LIN {X 0,Y 174.625,Z 737.69,A -85,B 0,C 180,E1 -22967.571,E2 -22967.571} C_VEL
LIN {X 0,Y 177.155,Z 732.813,A -85,B 0,C 180,E1 -22970.922,E2 -22970.922} C_VEL
LIN {X 0,Y 180.721,Z 725.647,A -85,B 0,C 180,E1 -22974.715,E2 -22974.715} C_VEL
LIN {X 0,Y 184.412,Z 717.918,A -85,B 0,C 180,E1 -22977.833,E2 -22977.833} C_VEL
LIN {X 0,Y 188.002,Z 709.609,A -85,B 0,C 180,E1 -22980.502,E2 -22980.502} C_VEL
LIN {X 0,Y 191.718,Z 699.712,A -85,B 0,C 180,E1 -22983.047,E2 -22983.047} C_VEL
LIN {X 0,Y 195.336,Z 689.177,A -85,B 0,C 180,E1 -22985.149,E2 -22985.149} C_VEL
LIN {X 0,Y 198.828,Z 677.532,A -85,B 0,C 180,E1 -22986.937,E2 -22986.937} C_VEL
LIN {X 0,Y 201.663,Z 665.358,A -85,B 0,C 180,E1 -22988.375,E2 -22988.375} C_VEL
LIN {X 0,Y 203.93,Z 652.017,A -85,B 0,C 180,E1 -22989.533,E2 -22989.533} C_VEL
LIN {X 0,Y 205.572,Z 638.845,A -85,B 0,C 180,E1 -22990.27,E2 -22990.27} C_VEL
LIN {X 0,Y 207.434,Z 606.957,A -85,B 0,C 180,E1 -22991.301,E2 -22991.301} C_VEL
LIN {X 0,Y 209.301,Z 573.723,A -85,B 0,C 180,E1 -22992.296,E2 -22992.296} C_VEL
LIN {X 0,Y 203.768,Z 561.065,A -85,B 0,C 180,E1 -22994.409,E2 -22994.409} C_VEL
LIN {X 0,Y 198.485,Z 550.546,A -85,B 0,C 180,E1 -22996.546,E2 -22996.546} C_VEL
LIN {X 0,Y 193.676,Z 542.168,A -85,B 0,C 180,E1 -22998.615,E2 -22998.615} C_VEL
LIN {X 0,Y 188.587,Z 533.88,A -85,B 0,C 180,E1 -23001.001,E2 -23001.001} C_VEL
LIN {X 0,Y 185.215,Z 528.789,A -85,B 0,C 180,E1 -23002.712,E2 -23002.712} C_VEL
LIN {X 0,Y 182.766,Z 526.441,A -85,B 0,C 180,E1 -23003.951,E2 -23003.951} C_VEL
LIN {X 0,Y 181.44,Z 526.477,A -85,B 0,C 180,E1 -23004.562,E2 -23004.562} C_VEL
LIN {X 0,Y 179.513,Z 527.597,A -85,B 0,C 180,E1 -23005.411,E2 -23005.411} C_VEL
LIN {X 0,Y 178.103,Z 527.429,A -85,B 0,C 180,E1 -23006.127,E2 -23006.127} C_VEL
LIN {X 0,Y 177.235,Z 526.122,A -85,B 0,C 180,E1 -23006.67,E2 -23006.67} C_VEL
LIN {X 0,Y 177.165,Z 525.886,A -85,B 0,C 180,E1 -23006.773,E2 -23006.773} C_VEL
LIN {X 0,Y 178.738,Z 533.065,A -85,B 0,C 180,E1 -23008.93,E2 -23008.93} C_VEL
LIN {X 0,Y 178.13,Z 538.271,A -85,B 0,C 180,E1 -23010.359,E2 -23010.359} C_VEL
LIN {X 0,Y 179.144,Z 556.855,A -85,B 0,C 180,E1 -23011.764,E2 -23011.764} C_VEL
LIN {X 0,Y 180.203,Z 569.633,A -85,B 0,C 180,E1 -23012.725,E2 -23012.725} C_VEL
LIN {X 0,Y 175.84,Z 649.181,A -85,B 0,C 180,E1 -23018.533,E2 -23018.533} C_VEL
LIN {X 0,Y 174.96,Z 664.149,A -85,B 0,C 180,E1 -23020.035,E2 -23020.035} C_VEL
LIN {X 0,Y 173.957,Z 676.673,A -85,B 0,C 180,E1 -23021.753,E2 -23021.753} C_VEL
LIN {X 0,Y 172.988,Z 688.326,A -85,B 0,C 180,E1 -23023.78,E2 -23023.78} C_VEL
LIN {X 0,Y 171.856,Z 700.346,A -85,B 0,C 180,E1 -23026.399,E2 -23026.399} C_VEL
LIN {X 0,Y 171.016,Z 711.334,A -85,B 0,C 180,E1 -23029.343,E2 -23029.343} C_VEL
LIN {X 0,Y 170.247,Z 721.958,A -85,B 0,C 180,E1 -23032.886,E2 -23032.886} C_VEL
LIN {X 0,Y 169.806,Z 730.545,A -85,B 0,C 180,E1 -23036.44,E2 -23036.44} C_VEL
LIN {X 0,Y 169.629,Z 737.453,A -85,B 0,C 180,E1 -23040,E2 -23040} C_VEL
LIN {X 0,Y 169.771,Z 743.094,A -85,B 0,C 180,E1 -23043.56,E2 -23043.56} C_VEL
LIN {X 0,Y 170.413,Z 748.728,A -85,B 0,C 180,E1 -23048.18,E2 -23048.18} C_VEL
LIN {X 0,Y 171.916,Z 752.123,A -85,B 0,C 180,E1 -23051.794,E2 -23051.794} C_VEL
LIN {X 0,Y 174.709,Z 755.167,A -85,B 0,C 180,E1 -23056.355,E2 -23056.355} C_VEL
LIN {X 0,Y 178.739,Z 756.761,A -85,B 0,C 180,E1 -23060.725,E2 -23060.725} C_VEL
LIN {X 0,Y 184.022,Z 756.991,A -85,B 0,C 180,E1 -23064.841,E2 -23064.841} C_VEL
LIN {X 0,Y 190.523,Z 755.83,A -85,B 0,C 180,E1 -23068.655,E2 -23068.655} C_VEL
LIN {X 0,Y 198.014,Z 753.226,A -85,B 0,C 180,E1 -23072.167,E2 -23072.167} C_VEL
LIN {X 0,Y 206.463,Z 749.156,A -85,B 0,C 180,E1 -23075.357,E2 -23075.357} C_VEL
LIN {X 0,Y 215.727,Z 743.443,A -85,B 0,C 180,E1 -23078.242,E2 -23078.242} C_VEL
LIN {X 0,Y 224.369,Z 737.019,A -85,B 0,C 180,E1 -23080.538,E2 -23080.538} C_VEL
LIN {X 0,Y 232.755,Z 729.734,A -85,B 0,C 180,E1 -23082.459,E2 -23082.459} C_VEL
LIN {X 0,Y 231.616,Z 730.78,A -85,B 0,C 180,E1 -23082.542,E2 -23082.542} C_VEL
LIN {X 0,Y 227.376,Z 734.465,A -85,B 0,C 180,E1 -23082.214,E2 -23082.214} C_VEL
LIN {X 0,Y 221.952,Z 738.733,A -85,B 0,C 180,E1 -23081.509,E2 -23081.509} C_VEL
LIN {X 0,Y 215.639,Z 743.149,A -85,B 0,C 180,E1 -23080.5,E2 -23080.5} C_VEL
LIN {X 0,Y 209.72,Z 746.748,A -85,B 0,C 180,E1 -23079.156,E2 -23079.156} C_VEL
LIN {X 0,Y 200.95,Z 751.371,A -85,B 0,C 180,E1 -23076.481,E2 -23076.481} C_VEL
LIN {X 0,Y 192.198,Z 754.859,A -85,B 0,C 180,E1 -23073.264,E2 -23073.264} C_VEL
LIN {X 0,Y 184.41,Z 756.936,A -85,B 0,C 180,E1 -23069.699,E2 -23069.699} C_VEL
LIN {X 0,Y 177.647,Z 757.638,A -85,B 0,C 180,E1 -23065.796,E2 -23065.796} C_VEL
LIN {X 0,Y 172.138,Z 756.939,A -85,B 0,C 180,E1 -23061.558,E2 -23061.558} C_VEL
LIN {X 0,Y 167.92,Z 754.893,A -85,B 0,C 180,E1 -23057.036,E2 -23057.036} C_VEL
LIN {X 0,Y 164.999,Z 751.477,A -85,B 0,C 180,E1 -23052.296,E2 -23052.296} C_VEL
LIN {X 0,Y 163.205,Z 746.501,A -85,B 0,C 180,E1 -23047.422,E2 -23047.422} C_VEL
LIN {X 0,Y 162.813,Z 741.678,A -85,B 0,C 180,E1 -23043.712,E2 -23043.712} C_VEL
LIN {X 0,Y 162.744,Z 734.637,A -85,B 0,C 180,E1 -23039.381,E2 -23039.381} C_VEL
LIN {X 0,Y 162.952,Z 727.007,A -85,B 0,C 180,E1 -23035.671,E2 -23035.671} C_VEL
LIN {X 0,Y 163.48,Z 717.634,A -85,B 0,C 180,E1 -23031.979,E2 -23031.979} C_VEL
LIN {X 0,Y 164.146,Z 708.066,A -85,B 0,C 180,E1 -23028.891,E2 -23028.891} C_VEL
LIN {X 0,Y 165.16,Z 696.327,A -85,B 0,C 180,E1 -23025.837,E2 -23025.837} C_VEL
LIN {X 0,Y 166.231,Z 684.876,A -85,B 0,C 180,E1 -23023.418,E2 -23023.418} C_VEL
LIN {X 0,Y 167.404,Z 670.266,A -85,B 0,C 180,E1 -23021.012,E2 -23021.012} C_VEL
LIN {X 0,Y 168.431,Z 655.646,A -85,B 0,C 180,E1 -23019.226,E2 -23019.226} C_VEL
LIN {X 0,Y 169.69,Z 632.143,A -85,B 0,C 180,E1 -23017.232,E2 -23017.232} C_VEL
LIN {X 0,Y 173.149,Z 568.211,A -85,B 0,C 180,E1 -23012.38,E2 -23012.38} C_VEL
LIN {X 0,Y 171.204,Z 544.253,A -85,B 0,C 180,E1 -23010.488,E2 -23010.488} C_VEL
LIN {X 0,Y 171.16,Z 538.339,A -85,B 0,C 180,E1 -23009.964,E2 -23009.964} C_VEL
LIN {X 0,Y 171.535,Z 535.378,A -85,B 0,C 180,E1 -23009.127,E2 -23009.127} C_VEL
LIN {X 0,Y 172.007,Z 536.683,A -85,B 0,C 180,E1 -23008.737,E2 -23008.737} C_VEL
LIN {X 0,Y 173.751,Z 536.615,A -85,B 0,C 180,E1 -23007.749,E2 -23007.749} C_VEL
LIN {X 0,Y 175.596,Z 535.684,A -85,B 0,C 180,E1 -23006.819,E2 -23006.819} C_VEL
LIN {X 0,Y 176.931,Z 534.47,A -85,B 0,C 180,E1 -23006.213,E2 -23006.213} C_VEL
LIN {X 0,Y 179.303,Z 534.57,A -85,B 0,C 180,E1 -23005.023,E2 -23005.023} C_VEL
LIN {X 0,Y 181.451,Z 533.728,A -85,B 0,C 180,E1 -23004.065,E2 -23004.065} C_VEL
LIN {X 0,Y 183.271,Z 536.04,A -85,B 0,C 180,E1 -23003.09,E2 -23003.09} C_VEL
LIN {X 0,Y 187.107,Z 542.192,A -85,B 0,C 180,E1 -23001.091,E2 -23001.091} C_VEL
LIN {X 0,Y 193.421,Z 553.044,A -85,B 0,C 180,E1 -22998.107,E2 -22998.107} C_VEL
LIN {X 0,Y 198.962,Z 564.124,A -85,B 0,C 180,E1 -22995.705,E2 -22995.705} C_VEL
LIN {X 0,Y 204.149,Z 576.218,A -85,B 0,C 180,E1 -22993.582,E2 -22993.582} C_VEL
LIN {X 0,Y 200.476,Z 637.51,A -85,B 0,C 180,E1 -22991.684,E2 -22991.684} C_VEL
LIN {X 0,Y 198.782,Z 651.222,A -85,B 0,C 180,E1 -22990.936,E2 -22990.936} C_VEL
LIN {X 0,Y 196.394,Z 664.844,A -85,B 0,C 180,E1 -22989.77,E2 -22989.77} C_VEL
LIN {X 0,Y 193.644,Z 676.37,A -85,B 0,C 180,E1 -22988.431,E2 -22988.431} C_VEL
LIN {X 0,Y 190.082,Z 688.373,A -85,B 0,C 180,E1 -22986.601,E2 -22986.601} C_VEL
LIN {X 0,Y 186.227,Z 699.112,A -85,B 0,C 180,E1 -22984.481,E2 -22984.481} C_VEL
LIN {X 0,Y 182.185,Z 709.349,A -85,B 0,C 180,E1 -22981.846,E2 -22981.846} C_VEL
LIN {X 0,Y 178.177,Z 718.346,A -85,B 0,C 180,E1 -22978.897,E2 -22978.897} C_VEL
LIN {X 0,Y 174.32,Z 726.066,A -85,B 0,C 180,E1 -22975.687,E2 -22975.687} C_VEL
LIN {X 0,Y 171.574,Z 731.344,A -85,B 0,C 180,E1 -22972.904,E2 -22972.904} C_VEL
LIN {X 0,Y 168.716,Z 736.585,A -85,B 0,C 180,E1 -22969.469,E2 -22969.469} C_VEL
LIN {X 0,Y 166.386,Z 740.746,A -85,B 0,C 180,E1 -22965.939,E2 -22965.939} C_VEL
LIN {X 0,Y 164.664,Z 743.938,A -85,B 0,C 180,E1 -22962.325,E2 -22962.325} C_VEL
LIN {X 0,Y 163.193,Z 746.789,A -85,B 0,C 180,E1 -22957.426,E2 -22957.426} C_VEL
LIN {X 0,Y 162.506,Z 748.203,A -85,B 0,C 180,E1 -22952.482,E2 -22952.482} C_VEL
LIN {X 0,Y 162.506,Z 748.173,A -85,B 0,C 180,E1 -22947.525,E2 -22947.525} C_VEL
LIN {X 0,Y 163.203,Z 746.722,A -85,B 0,C 180,E1 -22942.581,E2 -22942.581} C_VEL
LIN {X 0,Y 164.66,Z 743.832,A -85,B 0,C 180,E1 -22937.681,E2 -22937.681} C_VEL
LIN {X 0,Y 166.388,Z 740.593,A -85,B 0,C 180,E1 -22934.068,E2 -22934.068} C_VEL
LIN {X 0,Y 168.766,Z 736.381,A -85,B 0,C 180,E1 -22930.544,E2 -22930.544} C_VEL
LIN {X 0,Y 172.214,Z 730.105,A -85,B 0,C 180,E1 -22926.557,E2 -22926.557} C_VEL
LIN {X 0,Y 175.606,Z 723.348,A -85,B 0,C 180,E1 -22923.245,E2 -22923.245} C_VEL
LIN {X 0,Y 179.623,Z 715.035,A -85,B 0,C 180,E1 -22920.079,E2 -22920.079} C_VEL
LIN {X 0,Y 183.175,Z 706.616,A -85,B 0,C 180,E1 -22917.514,E2 -22917.514} C_VEL
LIN {X 0,Y 187.155,Z 696.339,A -85,B 0,C 180,E1 -22915.068,E2 -22915.068} C_VEL
LIN {X 0,Y 191.053,Z 684.888,A -85,B 0,C 180,E1 -22912.965,E2 -22912.965} C_VEL
LIN {X 0,Y 194.204,Z 673.731,A -85,B 0,C 180,E1 -22911.376,E2 -22911.376} C_VEL
LIN {X 0,Y 196.956,Z 661.448,A -85,B 0,C 180,E1 -22910.041,E2 -22910.041} C_VEL
LIN {X 0,Y 198.956,Z 648.868,A -85,B 0,C 180,E1 -22909.03,E2 -22909.03} C_VEL
LIN {X 0,Y 200.388,Z 636.086,A -85,B 0,C 180,E1 -22908.385,E2 -22908.385} C_VEL
LIN {X 0,Y 203.966,Z 575.937,A -85,B 0,C 180,E1 -22906.528,E2 -22906.528} C_VEL
LIN {X 0,Y 199.234,Z 564.909,A -85,B 0,C 180,E1 -22904.604,E2 -22904.604} C_VEL
LIN {X 0,Y 194.221,Z 554.656,A -85,B 0,C 180,E1 -22902.45,E2 -22902.45} C_VEL
LIN {X 0,Y 188.205,Z 544.028,A -85,B 0,C 180,E1 -22899.662,E2 -22899.662} C_VEL
LIN {X 0,Y 184.27,Z 537.742,A -85,B 0,C 180,E1 -22897.673,E2 -22897.673} C_VEL
LIN {X 0,Y 181.677,Z 533.791,A -85,B 0,C 180,E1 -22896.27,E2 -22896.27} C_VEL
LIN {X 0,Y 178.761,Z 529.44,A -85,B 0,C 180,E1 -22894.584,E2 -22894.584} C_VEL
LIN {X 0,Y 174.801,Z 524.016,A -85,B 0,C 180,E1 -22892.106,E2 -22892.106} C_VEL
LIN {X 0,Y 170.855,Z 518.693,A -85,B 0,C 180,E1 -22889.304,E2 -22889.304} C_VEL
LIN {X 0,Y 170.257,Z 516.653,A -85,B 0,C 180,E1 -22887.005,E2 -22887.005} C_VEL
LIN {X 0,Y 168.925,Z 513.033,A -85,B 0,C 180,E1 -22881.99,E2 -22881.99} C_VEL
LIN {X 0,Y 167.9,Z 510.255,A -85,B 0,C 180,E1 -22877.039,E2 -22877.039} C_VEL
LIN {X 0,Y 167.59,Z 509.067,A -85,B 0,C 180,E1 -22874.573,E2 -22874.573} C_VEL
LIN {X 0,Y 167.007,Z 507.441,A -85,B 0,C 180,E1 -22869.691,E2 -22869.691} C_VEL
LIN {X 0,Y 166.674,Z 506.615,A -85,B 0,C 180,E1 -22864.838,E2 -22864.838} C_VEL
LIN {X 0,Y 167.103,Z 506.205,A -85,B 0,C 180,E1 -22860,E2 -22860} C_VEL
LIN {X 0,Y 167.272,Z 507.771,A -85,B 0,C 180,E1 -22852.759,E2 -22852.759} C_VEL
LIN {X 0,Y 167.658,Z 508.512,A -85,B 0,C 180,E1 -22850.348,E2 -22850.348} C_VEL
LIN {X 0,Y 168.233,Z 510.934,A -85,B 0,C 180,E1 -22845.484,E2 -22845.484} C_VEL
LIN {X 0,Y 169.371,Z 513.991,A -85,B 0,C 180,E1 -22840.613,E2 -22840.613} C_VEL
LIN {X 0,Y 170.834,Z 517.869,A -85,B 0,C 180,E1 -22835.708,E2 -22835.708} C_VEL
LIN {X 0,Y 171.757,Z 520.239,A -85,B 0,C 180,E1 -22833.25,E2 -22833.25} C_VEL
LIN {X 0,Y 175.185,Z 525.109,A -85,B 0,C 180,E1 -22830.847,E2 -22830.847} C_VEL
LIN {X 0,Y 177.172,Z 527.91,A -85,B 0,C 180,E1 -22829.571,E2 -22829.571} C_VEL
LIN {X 0,Y 180.664,Z 532.795,A -85,B 0,C 180,E1 -22827.499,E2 -22827.499} C_VEL
LIN {X 0,Y 184.602,Z 538.886,A -85,B 0,C 180,E1 -22825.336,E2 -22825.336} C_VEL
LIN {X 0,Y 189.61,Z 547.065,A -85,B 0,C 180,E1 -22822.825,E2 -22822.825} C_VEL
LIN {X 0,Y 195.76,Z 558.495,A -85,B 0,C 180,E1 -22819.999,E2 -22819.999} C_VEL
LIN {X 0,Y 201.425,Z 570.829,A -85,B 0,C 180,E1 -22817.57,E2 -22817.57} C_VEL
LIN {X 0,Y 204.302,Z 577.81,A -85,B 0,C 180,E1 -22816.391,E2 -22816.391} C_VEL
LIN {X 0,Y 199.532,Z 648.468,A -85,B 0,C 180,E1 -22814.074,E2 -22814.074} C_VEL
LIN {X 0,Y 197.647,Z 662.676,A -85,B 0,C 180,E1 -22813.279,E2 -22813.279} C_VEL
LIN {X 0,Y 194.906,Z 676.278,A -85,B 0,C 180,E1 -22812.186,E2 -22812.186} C_VEL
LIN {X 0,Y 191.94,Z 688.053,A -85,B 0,C 180,E1 -22810.878,E2 -22810.878} C_VEL
LIN {X 0,Y 188.148,Z 700.496,A -85,B 0,C 180,E1 -22809.071,E2 -22809.071} C_VEL
LIN {X 0,Y 184.177,Z 711.686,A -85,B 0,C 180,E1 -22806.965,E2 -22806.965} C_VEL
LIN {X 0,Y 180.136,Z 722.07,A -85,B 0,C 180,E1 -22804.448,E2 -22804.448} C_VEL
LIN {X 0,Y 175.774,Z 732.205,A -85,B 0,C 180,E1 -22801.314,E2 -22801.314} C_VEL
LIN {X 0,Y 171.926,Z 740.549,A -85,B 0,C 180,E1 -22798.037,E2 -22798.037} C_VEL
LIN {X 0,Y 168.302,Z 748.481,A -85,B 0,C 180,E1 -22794.022,E2 -22794.022} C_VEL
LIN {X 0,Y 165.449,Z 754.781,A -85,B 0,C 180,E1 -22789.863,E2 -22789.863} C_VEL
LIN {X 0,Y 163.799,Z 759.021,A -85,B 0,C 180,E1 -22786.19,E2 -22786.19} C_VEL
LIN {X 0,Y 162.651,Z 762.322,A -85,B 0,C 180,E1 -22782.473,E2 -22782.473} C_VEL
LIN {X 0,Y 162.038,Z 765.357,A -85,B 0,C 180,E1 -22777.473,E2 -22777.473} C_VEL
LIN {X 0,Y 162.079,Z 766.544,A -85,B 0,C 180,E1 -22774.2,E2 -22774.2} C_VEL
LIN {X 0,Y 162.315,Z 767.113,A -85,B 0,C 180,E1 -22769.997,E2 -22769.997} C_VEL
LIN {X 0,Y 162.139,Z 766.498,A -85,B 0,C 180,E1 -22765.519,E2 -22765.519} C_VEL
LIN {X 0,Y 162.27,Z 765.398,A -85,B 0,C 180,E1 -22762.531,E2 -22762.531} C_VEL
LIN {X 0,Y 163.431,Z 762.363,A -85,B 0,C 180,E1 -22757.265,E2 -22757.265} C_VEL
LIN {X 0,Y 165.002,Z 764.433,A -85,B 0,C 180,E1 -22752.65,E2 -22752.65} C_VEL
LIN {X 0,Y 168.148,Z 765.424,A -85,B 0,C 180,E1 -22747.9,E2 -22747.9} C_VEL
LIN {X 0,Y 172.661,Z 765.196,A -85,B 0,C 180,E1 -22743.398,E2 -22743.398} C_VEL
LIN {X 0,Y 178.534,Z 763.777,A -85,B 0,C 180,E1 -22739.217,E2 -22739.217} C_VEL
LIN {X 0,Y 185.638,Z 761.165,A -85,B 0,C 180,E1 -22735.394,E2 -22735.394} C_VEL
LIN {X 0,Y 193.925,Z 757.314,A -85,B 0,C 180,E1 -22731.966,E2 -22731.966} C_VEL
LIN {X 0,Y 203.278,Z 752.1,A -85,B 0,C 180,E1 -22728.934,E2 -22728.934} C_VEL
LIN {X 0,Y 214.809,Z 744.407,A -85,B 0,C 180,E1 -22725.885,E2 -22725.885} C_VEL
LIN {X 0,Y 224.258,Z 737.146,A -85,B 0,C 180,E1 -22723.877,E2 -22723.877} C_VEL
LIN {X 0,Y 226.109,Z 735.546,A -85,B 0,C 180,E1 -22723.142,E2 -22723.142} C_VEL
LIN {X 0,Y 218.116,Z 741.451,A -85,B 0,C 180,E1 -22721.341,E2 -22721.341} C_VEL
LIN {X 0,Y 209.72,Z 746.748,A -85,B 0,C 180,E1 -22719.156,E2 -22719.156} C_VEL
LIN {X 0,Y 205.509,Z 749.08,A -85,B 0,C 180,E1 -22718.191,E2 -22718.191} C_VEL
LIN {X 0,Y 194.269,Z 753.932,A -85,B 0,C 180,E1 -22716.317,E2 -22716.317} C_VEL
LIN {X 0,Y 189.598,Z 755.467,A -85,B 0,C 180,E1 -22715.349,E2 -22715.349} C_VEL
LIN {X 0,Y 185.588,Z 756.528,A -85,B 0,C 180,E1 -22714.092,E2 -22714.092} C_VEL
LIN {X 0,Y 178.334,Z 757.885,A -85,B 0,C 180,E1 -22710.818,E2 -22710.818} C_VEL
LIN {X 0,Y 171.304,Z 758.107,A -85,B 0,C 180,E1 -22706.826,E2 -22706.826} C_VEL
LIN {X 0,Y 165.56,Z 756.971,A -85,B 0,C 180,E1 -22702.46,E2 -22702.46} C_VEL
LIN {X 0,Y 161.167,Z 754.483,A -85,B 0,C 180,E1 -22697.773,E2 -22697.773} C_VEL
LIN {X 0,Y 158.133,Z 750.643,A -85,B 0,C 180,E1 -22692.839,E2 -22692.839} C_VEL
LIN {X 0,Y 156.694,Z 747.057,A -85,B 0,C 180,E1 -22689.325,E2 -22689.325} C_VEL
LIN {X 0,Y 156,Z 741.962,A -85,B 0,C 180,E1 -22685.169,E2 -22685.169} C_VEL
LIN {X 0,Y 155.799,Z 734.936,A -85,B 0,C 180,E1 -22680.646,E2 -22680.646} C_VEL
LIN {X 0,Y 155.979,Z 727.459,A -85,B 0,C 180,E1 -22676.771,E2 -22676.771} C_VEL
LIN {X 0,Y 156.428,Z 718.366,A -85,B 0,C 180,E1 -22672.988,E2 -22672.988} C_VEL
LIN {X 0,Y 157.123,Z 708.727,A -85,B 0,C 180,E1 -22669.693,E2 -22669.693} C_VEL
LIN {X 0,Y 157.968,Z 697.197,A -85,B 0,C 180,E1 -22666.492,E2 -22666.492} C_VEL
LIN {X 0,Y 159.004,Z 685.993,A -85,B 0,C 180,E1 -22663.963,E2 -22663.963} C_VEL
LIN {X 0,Y 160.096,Z 672.673,A -85,B 0,C 180,E1 -22661.607,E2 -22661.607} C_VEL
LIN {X 0,Y 161.164,Z 658.975,A -85,B 0,C 180,E1 -22659.748,E2 -22659.748} C_VEL
LIN {X 0,Y 162.063,Z 642.966,A -85,B 0,C 180,E1 -22658.202,E2 -22658.202} C_VEL
LIN {X 0,Y 166.032,Z 568.178,A -85,B 0,C 180,E1 -22652.117,E2 -22652.117} C_VEL
LIN {X 0,Y 165.087,Z 558.183,A -85,B 0,C 180,E1 -22651.297,E2 -22651.297} C_VEL
LIN {X 0,Y 165.596,Z 559.295,A -85,B 0,C 180,E1 -22650.786,E2 -22650.786} C_VEL
LIN {X 0,Y 166.642,Z 559.167,A -85,B 0,C 180,E1 -22650.12,E2 -22650.12} C_VEL
LIN {X 0,Y 167.967,Z 557.129,A -85,B 0,C 180,E1 -22649.466,E2 -22649.466} C_VEL
LIN {X 0,Y 170.026,Z 551.583,A -85,B 0,C 180,E1 -22648.687,E2 -22648.687} C_VEL
LIN {X 0,Y 172.326,Z 543.836,A -85,B 0,C 180,E1 -22647.982,E2 -22647.982} C_VEL
LIN {X 0,Y 175.385,Z 542.887,A -85,B 0,C 180,E1 -22646.393,E2 -22646.393} C_VEL
LIN {X 0,Y 177.163,Z 541.617,A -85,B 0,C 180,E1 -22645.577,E2 -22645.577} C_VEL
LIN {X 0,Y 180.165,Z 541.5,A -85,B 0,C 180,E1 -22644.135,E2 -22644.135} C_VEL
LIN {X 0,Y 185.479,Z 550.34,A -85,B 0,C 180,E1 -22641.255,E2 -22641.255} C_VEL
LIN {X 0,Y 191.568,Z 561.63,A -85,B 0,C 180,E1 -22638.288,E2 -22638.288} C_VEL
LIN {X 0,Y 196.598,Z 572.5,A -85,B 0,C 180,E1 -22636.023,E2 -22636.023} C_VEL
LIN {X 0,Y 198.994,Z 578.319,A -85,B 0,C 180,E1 -22634.987,E2 -22634.987} C_VEL
LIN {X 0,Y 195.259,Z 638.519,A -85,B 0,C 180,E1 -22633.062,E2 -22633.062} C_VEL
LIN {X 0,Y 193.501,Z 651.963,A -85,B 0,C 180,E1 -22632.307,E2 -22632.307} C_VEL
LIN {X 0,Y 191.027,Z 665.457,A -85,B 0,C 180,E1 -22631.123,E2 -22631.123} C_VEL
LIN {X 0,Y 188.154,Z 676.913,A -85,B 0,C 180,E1 -22629.77,E2 -22629.77} C_VEL
LIN {X 0,Y 184.453,Z 688.854,A -85,B 0,C 180,E1 -22627.911,E2 -22627.911} C_VEL
LIN {X 0,Y 180.433,Z 699.569,A -85,B 0,C 180,E1 -22625.754,E2 -22625.754} C_VEL
LIN {X 0,Y 176.062,Z 710.141,A -85,B 0,C 180,E1 -22622.955,E2 -22622.955} C_VEL
LIN {X 0,Y 172.015,Z 718.774,A -85,B 0,C 180,E1 -22620.036,E2 -22620.036} C_VEL
LIN {X 0,Y 167.962,Z 726.486,A -85,B 0,C 180,E1 -22616.735,E2 -22616.735} C_VEL
LIN {X 0,Y 165.051,Z 731.76,A -85,B 0,C 180,E1 -22613.864,E2 -22613.864} C_VEL
LIN {X 0,Y 162.063,Z 736.996,A -85,B 0,C 180,E1 -22610.303,E2 -22610.303} C_VEL
LIN {X 0,Y 159.594,Z 741.155,A -85,B 0,C 180,E1 -22606.636,E2 -22606.636} C_VEL
LIN {X 0,Y 157.757,Z 744.345,A -85,B 0,C 180,E1 -22602.874,E2 -22602.874} C_VEL
LIN {X 0,Y 156.177,Z 747.197,A -85,B 0,C 180,E1 -22597.762,E2 -22597.762} C_VEL
LIN {X 0,Y 155.431,Z 748.611,A -85,B 0,C 180,E1 -22592.595,E2 -22592.595} C_VEL
LIN {X 0,Y 155.432,Z 748.582,A -85,B 0,C 180,E1 -22587.412,E2 -22587.412} C_VEL
LIN {X 0,Y 156.175,Z 747.132,A -85,B 0,C 180,E1 -22582.245,E2 -22582.245} C_VEL
LIN {X 0,Y 157.752,Z 744.241,A -85,B 0,C 180,E1 -22577.133,E2 -22577.133} C_VEL
LIN {X 0,Y 159.597,Z 741.003,A -85,B 0,C 180,E1 -22573.371,E2 -22573.371} C_VEL
LIN {X 0,Y 162.108,Z 736.794,A -85,B 0,C 180,E1 -22569.71,E2 -22569.71} C_VEL
LIN {X 0,Y 165.731,Z 730.523,A -85,B 0,C 180,E1 -22565.581,E2 -22565.581} C_VEL
LIN {X 0,Y 169.322,Z 723.771,A -85,B 0,C 180,E1 -22562.167,E2 -22562.167} C_VEL
LIN {X 0,Y 173.528,Z 715.472,A -85,B 0,C 180,E1 -22558.914,E2 -22558.914} C_VEL
LIN {X 0,Y 177.249,Z 707.067,A -85,B 0,C 180,E1 -22556.286,E2 -22556.286} C_VEL
LIN {X 0,Y 181.409,Z 696.814,A -85,B 0,C 180,E1 -22553.79,E2 -22553.79} C_VEL
LIN {X 0,Y 185.465,Z 685.394,A -85,B 0,C 180,E1 -22551.651,E2 -22551.651} C_VEL
LIN {X 0,Y 188.746,Z 674.285,A -85,B 0,C 180,E1 -22550.04,E2 -22550.04} C_VEL
LIN {X 0,Y 191.604,Z 662.077,A -85,B 0,C 180,E1 -22548.686,E2 -22548.686} C_VEL
LIN {X 0,Y 193.808,Z 648.811,A -85,B 0,C 180,E1 -22547.607,E2 -22547.607} C_VEL
LIN {X 0,Y 195.301,Z 635.824,A -85,B 0,C 180,E1 -22546.957,E2 -22546.957} C_VEL
LIN {X 0,Y 198.901,Z 578.234,A -85,B 0,C 180,E1 -22545.164,E2 -22545.164} C_VEL
LIN {X 0,Y 193.787,Z 566.354,A -85,B 0,C 180,E1 -22542.925,E2 -22542.925} C_VEL
LIN {X 0,Y 188.941,Z 556.662,A -85,B 0,C 180,E1 -22540.677,E2 -22540.677} C_VEL
LIN {X 0,Y 182.543,Z 545.353,A -85,B 0,C 180,E1 -22537.416,E2 -22537.416} C_VEL
LIN {X 0,Y 178.331,Z 538.872,A -85,B 0,C 180,E1 -22535.041,E2 -22535.041} C_VEL
LIN {X 0,Y 175.938,Z 535.201,A -85,B 0,C 180,E1 -22533.571,E2 -22533.571} C_VEL
LIN {X 0,Y 172.248,Z 529.975,A -85,B 0,C 180,E1 -22531.123,E2 -22531.123} C_VEL
LIN {X 0,Y 168.005,Z 524.32,A -85,B 0,C 180,E1 -22527.937,E2 -22527.937} C_VEL
LIN {X 0,Y 163.723,Z 518.755,A -85,B 0,C 180,E1 -22524.018,E2 -22524.018} C_VEL
LIN {X 0,Y 162.908,Z 516.336,A -85,B 0,C 180,E1 -22520.19,E2 -22520.19} C_VEL
LIN {X 0,Y 162.085,Z 513.767,A -85,B 0,C 180,E1 -22515.08,E2 -22515.08} C_VEL
LIN {X 0,Y 161.519,Z 512.038,A -85,B 0,C 180,E1 -22510.024,E2 -22510.024} C_VEL
LIN {X 0,Y 161.222,Z 511.162,A -85,B 0,C 180,E1 -22505.002,E2 -22505.002} C_VEL
LIN {X 0,Y 161.634,Z 510.777,A -85,B 0,C 180,E1 -22499.874,E2 -22499.874} C_VEL
LIN {X 0,Y 161.849,Z 512.376,A -85,B 0,C 180,E1 -22492.515,E2 -22492.515} C_VEL
LIN {X 0,Y 162.181,Z 513.194,A -85,B 0,C 180,E1 -22490.018,E2 -22490.018} C_VEL
LIN {X 0,Y 162.798,Z 515.667,A -85,B 0,C 180,E1 -22484.988,E2 -22484.988} C_VEL
LIN {X 0,Y 163.925,Z 518.88,A -85,B 0,C 180,E1 -22479.941,E2 -22479.941} C_VEL
LIN {X 0,Y 164.487,Z 520.164,A -85,B 0,C 180,E1 -22478.376,E2 -22478.376} C_VEL
LIN {X 0,Y 168.883,Z 525.83,A -85,B 0,C 180,E1 -22474.59,E2 -22474.59} C_VEL
LIN {X 0,Y 170.34,Z 527.932,A -85,B 0,C 180,E1 -22473.456,E2 -22473.456} C_VEL
LIN {X 0,Y 174.255,Z 533.373,A -85,B 0,C 180,E1 -22470.7,E2 -22470.7} C_VEL
LIN {X 0,Y 177.951,Z 538.843,A -85,B 0,C 180,E1 -22468.364,E2 -22468.364} C_VEL
LIN {X 0,Y 181.377,Z 544.285,A -85,B 0,C 180,E1 -22466.375,E2 -22466.375} C_VEL
LIN {X 0,Y 186.023,Z 552.086,A -85,B 0,C 180,E1 -22463.904,E2 -22463.904} C_VEL
LIN {X 0,Y 191.879,Z 563.306,A -85,B 0,C 180,E1 -22461.043,E2 -22461.043} C_VEL
LIN {X 0,Y 197.314,Z 575.454,A -85,B 0,C 180,E1 -22458.569,E2 -22458.569} C_VEL
LIN {X 0,Y 199.213,Z 580.128,A -85,B 0,C 180,E1 -22457.74,E2 -22457.74} C_VEL
LIN {X 0,Y 194.351,Z 648.588,A -85,B 0,C 180,E1 -22455.48,E2 -22455.48} C_VEL
LIN {X 0,Y 192.392,Z 662.677,A -85,B 0,C 180,E1 -22454.68,E2 -22454.68} C_VEL
LIN {X 0,Y 189.436,Z 676.777,A -85,B 0,C 180,E1 -22453.52,E2 -22453.52} C_VEL
LIN {X 0,Y 186.132,Z 689.272,A -85,B 0,C 180,E1 -22452.079,E2 -22452.079} C_VEL
LIN {X 0,Y 182.171,Z 701.377,A -85,B 0,C 180,E1 -22450.251,E2 -22450.251} C_VEL
LIN {X 0,Y 177.957,Z 712.651,A -85,B 0,C 180,E1 -22448.016,E2 -22448.016} C_VEL
LIN {X 0,Y 173.488,Z 723.429,A -85,B 0,C 180,E1 -22445.254,E2 -22445.254} C_VEL
LIN {X 0,Y 168.972,Z 733.28,A -85,B 0,C 180,E1 -22442.022,E2 -22442.022} C_VEL
LIN {X 0,Y 165.028,Z 741.379,A -85,B 0,C 180,E1 -22438.623,E2 -22438.623} C_VEL
LIN {X 0,Y 161.3,Z 749.07,A -85,B 0,C 180,E1 -22434.448,E2 -22434.448} C_VEL
LIN {X 0,Y 158.703,Z 754.359,A -85,B 0,C 180,E1 -22430.745,E2 -22430.745} C_VEL
LIN {X 0,Y 156.914,Z 758.603,A -85,B 0,C 180,E1 -22426.922,E2 -22426.922} C_VEL
LIN {X 0,Y 155.664,Z 761.907,A -85,B 0,C 180,E1 -22423.043,E2 -22423.043} C_VEL
LIN {X 0,Y 154.959,Z 764.944,A -85,B 0,C 180,E1 -22417.817,E2 -22417.817} C_VEL
LIN {X 0,Y 155.008,Z 766.197,A -85,B 0,C 180,E1 -22414.077,E2 -22414.077} C_VEL
LIN {X 0,Y 155.23,Z 766.704,A -85,B 0,C 180,E1 -22409.997,E2 -22409.997} C_VEL
LIN {X 0,Y 155.056,Z 766.164,A -85,B 0,C 180,E1 -22405.679,E2 -22405.679} C_VEL
LIN {X 0,Y 155.21,Z 764.987,A -85,B 0,C 180,E1 -22402.189,E2 -22402.189} C_VEL
LIN {X 0,Y 156.387,Z 761.995,A -85,B 0,C 180,E1 -22397.012,E2 -22397.012} C_VEL
LIN {X 0,Y 156.815,Z 761.321,A -85,B 0,C 180,E1 -22395.892,E2 -22395.892} C_VEL
LIN {X 0,Y 158.32,Z 763.244,A -85,B 0,C 180,E1 -22391.893,E2 -22391.893} C_VEL
LIN {X 0,Y 161.61,Z 764.62,A -85,B 0,C 180,E1 -22386.956,E2 -22386.956} C_VEL
LIN {X 0,Y 166.337,Z 764.821,A -85,B 0,C 180,E1 -22382.302,E2 -22382.302} C_VEL
LIN {X 0,Y 172.472,Z 763.864,A -85,B 0,C 180,E1 -22378.009,E2 -22378.009} C_VEL
LIN {X 0,Y 179.87,Z 761.746,A -85,B 0,C 180,E1 -22374.117,E2 -22374.117} C_VEL
LIN {X 0,Y 188.466,Z 758.437,A -85,B 0,C 180,E1 -22370.655,E2 -22370.655} C_VEL
LIN {X 0,Y 198.093,Z 753.846,A -85,B 0,C 180,E1 -22367.613,E2 -22367.613} C_VEL
LIN {X 0,Y 208.507,Z 747.872,A -85,B 0,C 180,E1 -22364.938,E2 -22364.938} C_VEL
LIN {X 0,Y 213.964,Z 744.358,A -85,B 0,C 180,E1 -22363.725,E2 -22363.725} C_VEL
LIN {X 0,Y 215.889,Z 743.057,A -85,B 0,C 180,E1 -22363.128,E2 -22363.128} C_VEL
LIN {X 0,Y 205.339,Z 749.013,A -85,B 0,C 180,E1 -22360.564,E2 -22360.564} C_VEL
LIN {X 0,Y 195.474,Z 753.435,A -85,B 0,C 180,E1 -22357.677,E2 -22357.677} C_VEL
LIN {X 0,Y 186.426,Z 756.342,A -85,B 0,C 180,E1 -22354.435,E2 -22354.435} C_VEL
LIN {X 0,Y 185.588,Z 756.528,A -85,B 0,C 180,E1 -22354.092,E2 -22354.092} C_VEL
LIN {X 0,Y 181.621,Z 757.425,A -85,B 0,C 180,E1 -22352.74,E2 -22352.74} C_VEL
LIN {X 0,Y 173.955,Z 758.399,A -85,B 0,C 180,E1 -22350.723,E2 -22350.723} C_VEL
LIN {X 0,Y 168.003,Z 758.574,A -85,B 0,C 180,E1 -22348.979,E2 -22348.979} C_VEL
LIN {X 0,Y 164.341,Z 758.291,A -85,B 0,C 180,E1 -22347.397,E2 -22347.397} C_VEL
LIN {X 0,Y 163.393,Z 758.072,A -85,B 0,C 180,E1 -22346.8,E2 -22346.8} C_VEL
LIN {X 0,Y 159.035,Z 756.821,A -85,B 0,C 180,E1 -22343.436,E2 -22343.436} C_VEL
LIN {X 0,Y 154.452,Z 753.913,A -85,B 0,C 180,E1 -22338.573,E2 -22338.573} C_VEL
LIN {X 0,Y 151.305,Z 749.618,A -85,B 0,C 180,E1 -22333.429,E2 -22333.429} C_VEL
LIN {X 0,Y 149.416,Z 743.838,A -85,B 0,C 180,E1 -22328.112,E2 -22328.112} C_VEL
LIN {X 0,Y 148.964,Z 737.322,A -85,B 0,C 180,E1 -22323.381,E2 -22323.381} C_VEL
LIN {X 0,Y 148.994,Z 730.389,A -85,B 0,C 180,E1 -22319.324,E2 -22319.324} C_VEL
LIN {X 0,Y 149.258,Z 721.814,A -85,B 0,C 180,E1 -22315.273,E2 -22315.273} C_VEL
LIN {X 0,Y 149.773,Z 713.221,A -85,B 0,C 180,E1 -22311.907,E2 -22311.907} C_VEL
LIN {X 0,Y 150.452,Z 703.159,A -85,B 0,C 180,E1 -22308.678,E2 -22308.678} C_VEL
LIN {X 0,Y 151.443,Z 691.184,A -85,B 0,C 180,E1 -22305.555,E2 -22305.555} C_VEL
LIN {X 0,Y 152.545,Z 678.49,A -85,B 0,C 180,E1 -22302.92,E2 -22302.92} C_VEL
LIN {X 0,Y 153.577,Z 665.472,A -85,B 0,C 180,E1 -22300.797,E2 -22300.797} C_VEL
LIN {X 0,Y 154.42,Z 652.119,A -85,B 0,C 180,E1 -22299.171,E2 -22299.171} C_VEL
LIN {X 0,Y 157.007,Z 601.86,A -85,B 0,C 180,E1 -22294.745,E2 -22294.745} C_VEL
LIN {X 0,Y 157.757,Z 588.664,A -85,B 0,C 180,E1 -22293.634,E2 -22293.634} C_VEL
LIN {X 0,Y 157.944,Z 591.261,A -85,B 0,C 180,E1 -22293.157,E2 -22293.157} C_VEL
LIN {X 0,Y 158.253,Z 591.635,A -85,B 0,C 180,E1 -22292.883,E2 -22292.883} C_VEL
LIN {X 0,Y 159.182,Z 590.427,A -85,B 0,C 180,E1 -22292.313,E2 -22292.313} C_VEL
LIN {X 0,Y 161.375,Z 584.884,A -85,B 0,C 180,E1 -22291.287,E2 -22291.287} C_VEL
LIN {X 0,Y 164.691,Z 573.851,A -85,B 0,C 180,E1 -22290.082,E2 -22290.082} C_VEL
LIN {X 0,Y 166.863,Z 566.025,A -85,B 0,C 180,E1 -22289.391,E2 -22289.391} C_VEL
LIN {X 0,Y 168.72,Z 564.138,A -85,B 0,C 180,E1 -22288.43,E2 -22288.43} C_VEL
LIN {X 0,Y 170.596,Z 560.816,A -85,B 0,C 180,E1 -22287.618,E2 -22287.618} C_VEL
LIN {X 0,Y 172.902,Z 554.909,A -85,B 0,C 180,E1 -22286.806,E2 -22286.806} C_VEL
LIN {X 0,Y 174.413,Z 550.255,A -85,B 0,C 180,E1 -22286.354,E2 -22286.354} C_VEL
LIN {X 0,Y 177.421,Z 548.722,A -85,B 0,C 180,E1 -22284.944,E2 -22284.944} C_VEL
LIN {X 0,Y 178.252,Z 548.957,A -85,B 0,C 180,E1 -22284.526,E2 -22284.526} C_VEL
LIN {X 0,Y 182.267,Z 555.807,A -85,B 0,C 180,E1 -22282.256,E2 -22282.256} C_VEL
LIN {X 0,Y 187.996,Z 566.801,A -85,B 0,C 180,E1 -22279.297,E2 -22279.297} C_VEL
LIN {X 0,Y 192.837,Z 577.656,A -85,B 0,C 180,E1 -22276.983,E2 -22276.983} C_VEL
LIN {X 0,Y 194.042,Z 580.735,A -85,B 0,C 180,E1 -22276.421,E2 -22276.421} C_VEL
LIN {X 0,Y 190.293,Z 638.353,A -85,B 0,C 180,E1 -22274.568,E2 -22274.568} C_VEL
LIN {X 0,Y 188.47,Z 651.934,A -85,B 0,C 180,E1 -22273.807,E2 -22273.807} C_VEL
LIN {X 0,Y 186.017,Z 664.942,A -85,B 0,C 180,E1 -22272.668,E2 -22272.668} C_VEL
LIN {X 0,Y 182.769,Z 677.456,A -85,B 0,C 180,E1 -22271.189,E2 -22271.189} C_VEL
LIN {X 0,Y 178.938,Z 689.333,A -85,B 0,C 180,E1 -22269.299,E2 -22269.299} C_VEL
LIN {X 0,Y 174.738,Z 700.025,A -85,B 0,C 180,E1 -22267.11,E2 -22267.11} C_VEL
LIN {X 0,Y 170.519,Z 709.819,A -85,B 0,C 180,E1 -22264.481,E2 -22264.481} C_VEL
LIN {X 0,Y 165.929,Z 719.202,A -85,B 0,C 180,E1 -22261.259,E2 -22261.259} C_VEL
LIN {X 0,Y 161.654,Z 726.907,A -85,B 0,C 180,E1 -22257.867,E2 -22257.867} C_VEL
LIN {X 0,Y 157.479,Z 734.051,A -85,B 0,C 180,E1 -22253.685,E2 -22253.685} C_VEL
LIN {X 0,Y 154.482,Z 738.92,A -85,B 0,C 180,E1 -22249.954,E2 -22249.954} C_VEL
LIN {X 0,Y 152.066,Z 742.758,A -85,B 0,C 180,E1 -22246.103,E2 -22246.103} C_VEL
LIN {X 0,Y 149.868,Z 746.366,A -85,B 0,C 180,E1 -22240.815,E2 -22240.815} C_VEL
LIN {X 0,Y 148.682,Z 748.487,A -85,B 0,C 180,E1 -22235.428,E2 -22235.428} C_VEL
LIN {X 0,Y 148.265,Z 749.191,A -85,B 0,C 180,E1 -22230.004,E2 -22230.004} C_VEL
LIN {X 0,Y 148.686,Z 748.44,A -85,B 0,C 180,E1 -22224.579,E2 -22224.579} C_VEL
LIN {X 0,Y 149.863,Z 746.282,A -85,B 0,C 180,E1 -22219.192,E2 -22219.192} C_VEL
LIN {X 0,Y 152.074,Z 742.621,A -85,B 0,C 180,E1 -22213.905,E2 -22213.905} C_VEL
LIN {X 0,Y 154.54,Z 738.745,A -85,B 0,C 180,E1 -22210.061,E2 -22210.061} C_VEL
LIN {X 0,Y 157.573,Z 733.827,A -85,B 0,C 180,E1 -22206.337,E2 -22206.337} C_VEL
LIN {X 0,Y 161.092,Z 727.742,A -85,B 0,C 180,E1 -22202.74,E2 -22202.74} C_VEL
LIN {X 0,Y 165.237,Z 720.266,A -85,B 0,C 180,E1 -22199.314,E2 -22199.314} C_VEL
LIN {X 0,Y 169.921,Z 710.928,A -85,B 0,C 180,E1 -22196.018,E2 -22196.018} C_VEL
LIN {X 0,Y 173.948,Z 701.619,A -85,B 0,C 180,E1 -22193.424,E2 -22193.424} C_VEL
LIN {X 0,Y 178.058,Z 691.272,A -85,B 0,C 180,E1 -22191.205,E2 -22191.205} C_VEL
LIN {X 0,Y 181.869,Z 679.899,A -85,B 0,C 180,E1 -22189.304,E2 -22189.304} C_VEL
LIN {X 0,Y 185.361,Z 667.189,A -85,B 0,C 180,E1 -22187.706,E2 -22187.706} C_VEL
LIN {X 0,Y 187.984,Z 654.259,A -85,B 0,C 180,E1 -22186.521,E2 -22186.521} C_VEL
LIN {X 0,Y 189.661,Z 641.912,A -85,B 0,C 180,E1 -22185.716,E2 -22185.716} C_VEL
LIN {X 0,Y 191.071,Z 624.209,A -85,B 0,C 180,E1 -22185.062,E2 -22185.062} C_VEL
LIN {X 0,Y 193.893,Z 580.536,A -85,B 0,C 180,E1 -22183.706,E2 -22183.706} C_VEL
LIN {X 0,Y 188.858,Z 568.71,A -85,B 0,C 180,E1 -22181.328,E2 -22181.328} C_VEL
LIN {X 0,Y 183.721,Z 558.593,A -85,B 0,C 180,E1 -22178.747,E2 -22178.747} C_VEL
LIN {X 0,Y 178.592,Z 549.596,A -85,B 0,C 180,E1 -22175.913,E2 -22175.913} C_VEL
LIN {X 0,Y 175.185,Z 544.063,A -85,B 0,C 180,E1 -22173.837,E2 -22173.837} C_VEL
LIN {X 0,Y 172.599,Z 540.137,A -85,B 0,C 180,E1 -22172.14,E2 -22172.14} C_VEL
LIN {X 0,Y 169.863,Z 536.099,A -85,B 0,C 180,E1 -22170.196,E2 -22170.196} C_VEL
LIN {X 0,Y 165.947,Z 530.63,A -85,B 0,C 180,E1 -22167.083,E2 -22167.083} C_VEL
LIN {X 0,Y 161.515,Z 524.99,A -85,B 0,C 180,E1 -22162.886,E2 -22162.886} C_VEL
LIN {X 0,Y 156.709,Z 518.927,A -85,B 0,C 180,E1 -22156.613,E2 -22156.613} C_VEL
LIN {X 0,Y 156.277,Z 517.446,A -85,B 0,C 180,E1 -22152.995,E2 -22152.995} C_VEL
LIN {X 0,Y 155.876,Z 515.977,A -85,B 0,C 180,E1 -22147.32,E2 -22147.32} C_VEL
LIN {X 0,Y 156.183,Z 515.31,A -85,B 0,C 180,E1 -22140,E2 -22140} C_VEL
LIN {X 0,Y 156.549,Z 517.41,A -85,B 0,C 180,E1 -22130.962,E2 -22130.962} C_VEL
LIN {X 0,Y 157.257,Z 519.937,A -85,B 0,C 180,E1 -22125.606,E2 -22125.606} C_VEL
LIN {X 0,Y 162.838,Z 527.021,A -85,B 0,C 180,E1 -22118.976,E2 -22118.976} C_VEL
LIN {X 0,Y 167.486,Z 533.127,A -85,B 0,C 180,E1 -22114.845,E2 -22114.845} C_VEL
LIN {X 0,Y 171.777,Z 539.474,A -85,B 0,C 180,E1 -22111.601,E2 -22111.601} C_VEL
LIN {X 0,Y 175.469,Z 545.162,A -85,B 0,C 180,E1 -22109.141,E2 -22109.141} C_VEL
LIN {X 0,Y 180.102,Z 552.779,A -85,B 0,C 180,E1 -22106.366,E2 -22106.366} C_VEL
LIN {X 0,Y 185.244,Z 562.402,A -85,B 0,C 180,E1 -22103.56,E2 -22103.56} C_VEL
LIN {X 0,Y 190.067,Z 572.552,A -85,B 0,C 180,E1 -22101.141,E2 -22101.141} C_VEL
LIN {X 0,Y 194.169,Z 582.349,A -85,B 0,C 180,E1 -22099.191,E2 -22099.191} C_VEL
LIN {X 0,Y 189.433,Z 647.58,A -85,B 0,C 180,E1 -22097.014,E2 -22097.014} C_VEL
LIN {X 0,Y 187.41,Z 661.924,A -85,B 0,C 180,E1 -22096.206,E2 -22096.206} C_VEL
LIN {X 0,Y 184.63,Z 675.019,A -85,B 0,C 180,E1 -22095.146,E2 -22095.146} C_VEL
LIN {X 0,Y 181.405,Z 686.937,A -85,B 0,C 180,E1 -22093.825,E2 -22093.825} C_VEL
LIN {X 0,Y 177.288,Z 699.471,A -85,B 0,C 180,E1 -22091.982,E2 -22091.982} C_VEL
LIN {X 0,Y 172.86,Z 711.055,A -85,B 0,C 180,E1 -22089.738,E2 -22089.738} C_VEL
LIN {X 0,Y 168.561,Z 721.17,A -85,B 0,C 180,E1 -22087.193,E2 -22087.193} C_VEL
LIN {X 0,Y 163.73,Z 731.331,A -85,B 0,C 180,E1 -22083.915,E2 -22083.915} C_VEL
LIN {X 0,Y 159.423,Z 739.69,A -85,B 0,C 180,E1 -22080.458,E2 -22080.458} C_VEL
LIN {X 0,Y 155.317,Z 747.632,A -85,B 0,C 180,E1 -22076.175,E2 -22076.175} C_VEL
LIN {X 0,Y 152.007,Z 753.938,A -85,B 0,C 180,E1 -22071.704,E2 -22071.704} C_VEL
LIN {X 0,Y 150.058,Z 758.185,A -85,B 0,C 180,E1 -22067.72,E2 -22067.72} C_VEL
LIN {X 0,Y 148.681,Z 761.491,A -85,B 0,C 180,E1 -22063.667,E2 -22063.667} C_VEL
LIN {X 0,Y 147.883,Z 764.531,A -85,B 0,C 180,E1 -22058.193,E2 -22058.193} C_VEL
LIN {X 0,Y 147.938,Z 765.85,A -85,B 0,C 180,E1 -22053.946,E2 -22053.946} C_VEL
LIN {X 0,Y 148.145,Z 766.296,A -85,B 0,C 180,E1 -22049.996,E2 -22049.996} C_VEL
LIN {X 0,Y 147.962,Z 765.84,A -85,B 0,C 180,E1 -22045.921,E2 -22045.921} C_VEL
LIN {X 0,Y 148.16,Z 764.576,A -85,B 0,C 180,E1 -22041.815,E2 -22041.815} C_VEL
LIN {X 0,Y 149.459,Z 761.585,A -85,B 0,C 180,E1 -22036.398,E2 -22036.398} C_VEL
LIN {X 0,Y 150.316,Z 760.197,A -85,B 0,C 180,E1 -22034.401,E2 -22034.401} C_VEL
LIN {X 0,Y 153.211,Z 762.934,A -85,B 0,C 180,E1 -22028.468,E2 -22028.468} C_VEL
LIN {X 0,Y 157.423,Z 764.12,A -85,B 0,C 180,E1 -22023.481,E2 -22023.481} C_VEL
LIN {X 0,Y 163.169,Z 764.182,A -85,B 0,C 180,E1 -22018.875,E2 -22018.875} C_VEL
LIN {X 0,Y 170.162,Z 763.114,A -85,B 0,C 180,E1 -22014.671,E2 -22014.671} C_VEL
LIN {X 0,Y 178.519,Z 760.919,A -85,B 0,C 180,E1 -22010.954,E2 -22010.954} C_VEL
LIN {X 0,Y 187.903,Z 757.558,A -85,B 0,C 180,E1 -22007.679,E2 -22007.679} C_VEL
LIN {X 0,Y 198.288,Z 752.911,A -85,B 0,C 180,E1 -22004.854,E2 -22004.854} C_VEL
LIN {X 0,Y 205.58,Z 749.094,A -85,B 0,C 180,E1 -22003.135,E2 -22003.135} C_VEL
LIN {X 0,Y 195.053,Z 753.599,A -85,B 0,C 180,E1 -22000.433,E2 -22000.433} C_VEL
LIN {X 0,Y 185.267,Z 756.674,A -85,B 0,C 180,E1 -21997.369,E2 -21997.369} C_VEL
LIN {X 0,Y 176.397,Z 758.338,A -85,B 0,C 180,E1 -21993.903,E2 -21993.903} C_VEL
LIN {X 0,Y 168.58,Z 758.701,A -85,B 0,C 180,E1 -21990.018,E2 -21990.018} C_VEL
LIN {X 0,Y 163.393,Z 758.072,A -85,B 0,C 180,E1 -21986.8,E2 -21986.8} C_VEL
LIN {X 0,Y 160.316,Z 757.466,A -85,B 0,C 180,E1 -21985.034,E2 -21985.034} C_VEL
LIN {X 0,Y 154.096,Z 755.777,A -85,B 0,C 180,E1 -21982.296,E2 -21982.296} C_VEL
LIN {X 0,Y 148.427,Z 753.229,A -85,B 0,C 180,E1 -21979.367,E2 -21979.367} C_VEL
LIN {X 0,Y 146.3,Z 751.422,A -85,B 0,C 180,E1 -21977.336,E2 -21977.336} C_VEL
LIN {X 0,Y 143.837,Z 746.893,A -85,B 0,C 180,E1 -21972.558,E2 -21972.558} C_VEL
LIN {X 0,Y 142.405,Z 740.376,A -85,B 0,C 180,E1 -21967.087,E2 -21967.087} C_VEL
LIN {X 0,Y 142.13,Z 734.141,A -85,B 0,C 180,E1 -21962.834,E2 -21962.834} C_VEL
LIN {X 0,Y 142.214,Z 726.539,A -85,B 0,C 180,E1 -21958.584,E2 -21958.584} C_VEL
LIN {X 0,Y 142.49,Z 718.844,A -85,B 0,C 180,E1 -21955.048,E2 -21955.048} C_VEL
LIN {X 0,Y 143.114,Z 708.531,A -85,B 0,C 180,E1 -21951.14,E2 -21951.14} C_VEL
LIN {X 0,Y 143.921,Z 696.951,A -85,B 0,C 180,E1 -21947.608,E2 -21947.608} C_VEL
LIN {X 0,Y 144.83,Z 685.972,A -85,B 0,C 180,E1 -21944.88,E2 -21944.88} C_VEL
LIN {X 0,Y 145.82,Z 673.716,A -85,B 0,C 180,E1 -21942.468,E2 -21942.468} C_VEL
LIN {X 0,Y 146.858,Z 660.501,A -85,B 0,C 180,E1 -21940.428,E2 -21940.428} C_VEL
LIN {X 0,Y 147.856,Z 643.587,A -85,B 0,C 180,E1 -21938.567,E2 -21938.567} C_VEL
LIN {X 0,Y 148.544,Z 628.275,A -85,B 0,C 180,E1 -21937.117,E2 -21937.117} C_VEL
LIN {X 0,Y 148.621,Z 630.837,A -85,B 0,C 180,E1 -21936.669,E2 -21936.669} C_VEL
LIN {X 0,Y 148.886,Z 631.414,A -85,B 0,C 180,E1 -21936.344,E2 -21936.344} C_VEL
LIN {X 0,Y 149.44,Z 630.958,A -85,B 0,C 180,E1 -21935.885,E2 -21935.885} C_VEL
LIN {X 0,Y 150.453,Z 628.77,A -85,B 0,C 180,E1 -21935.231,E2 -21935.231} C_VEL
LIN {X 0,Y 152.578,Z 622.322,A -85,B 0,C 180,E1 -21934.141,E2 -21934.141} C_VEL
LIN {X 0,Y 155.96,Z 609.88,A -85,B 0,C 180,E1 -21932.771,E2 -21932.771} C_VEL
LIN {X 0,Y 158.857,Z 598.105,A -85,B 0,C 180,E1 -21931.799,E2 -21931.799} C_VEL
LIN {X 0,Y 160.591,Z 595.999,A -85,B 0,C 180,E1 -21930.792,E2 -21930.792} C_VEL
LIN {X 0,Y 162.328,Z 592.485,A -85,B 0,C 180,E1 -21929.961,E2 -21929.961} C_VEL
LIN {X 0,Y 165.098,Z 584.907,A -85,B 0,C 180,E1 -21928.877,E2 -21928.877} C_VEL
LIN {X 0,Y 169.223,Z 571.078,A -85,B 0,C 180,E1 -21927.583,E2 -21927.583} C_VEL
LIN {X 0,Y 171.875,Z 567.476,A -85,B 0,C 180,E1 -21926.406,E2 -21926.406} C_VEL
LIN {X 0,Y 174.343,Z 562.413,A -85,B 0,C 180,E1 -21925.498,E2 -21925.498} C_VEL
LIN {X 0,Y 176.381,Z 556.845,A -85,B 0,C 180,E1 -21924.881,E2 -21924.881} C_VEL
LIN {X 0,Y 176.738,Z 556.926,A -85,B 0,C 180,E1 -21924.701,E2 -21924.701} C_VEL
LIN {X 0,Y 182.528,Z 567.884,A -85,B 0,C 180,E1 -21921.386,E2 -21921.386} C_VEL
LIN {X 0,Y 187.021,Z 577.768,A -85,B 0,C 180,E1 -21919.032,E2 -21919.032} C_VEL
LIN {X 0,Y 189.24,Z 583.171,A -85,B 0,C 180,E1 -21917.922,E2 -21917.922} C_VEL
LIN {X 0,Y 185.334,Z 639.342,A -85,B 0,C 180,E1 -21916.099,E2 -21916.099} C_VEL
LIN {X 0,Y 183.309,Z 653.436,A -85,B 0,C 180,E1 -21915.278,E2 -21915.278} C_VEL
LIN {X 0,Y 180.641,Z 666.682,A -85,B 0,C 180,E1 -21914.066,E2 -21914.066} C_VEL
LIN {X 0,Y 177.509,Z 677.996,A -85,B 0,C 180,E1 -21912.693,E2 -21912.693} C_VEL
LIN {X 0,Y 173.523,Z 689.813,A -85,B 0,C 180,E1 -21910.779,E2 -21910.779} C_VEL
LIN {X 0,Y 169.139,Z 700.482,A -85,B 0,C 180,E1 -21908.559,E2 -21908.559} C_VEL
LIN {X 0,Y 164.529,Z 710.676,A -85,B 0,C 180,E1 -21905.746,E2 -21905.746} C_VEL
LIN {X 0,Y 159.926,Z 719.629,A -85,B 0,C 180,E1 -21902.573,E2 -21902.573} C_VEL
LIN {X 0,Y 155.428,Z 727.325,A -85,B 0,C 180,E1 -21899.087,E2 -21899.087} C_VEL
LIN {X 0,Y 152.184,Z 732.59,A -85,B 0,C 180,E1 -21896.026,E2 -21896.026} C_VEL
LIN {X 0,Y 148.859,Z 737.818,A -85,B 0,C 180,E1 -21892.195,E2 -21892.195} C_VEL
LIN {X 0,Y 146.053,Z 741.975,A -85,B 0,C 180,E1 -21888.23,E2 -21888.23} C_VEL
LIN {X 0,Y 143.968,Z 745.162,A -85,B 0,C 180,E1 -21884.131,E2 -21884.131} C_VEL
LIN {X 0,Y 142.175,Z 748.012,A -85,B 0,C 180,E1 -21878.532,E2 -21878.532} C_VEL
LIN {X 0,Y 141.291,Z 749.428,A -85,B 0,C 180,E1 -21872.855,E2 -21872.855} C_VEL
LIN {X 0,Y 141.292,Z 749.4,A -85,B 0,C 180,E1 -21867.153,E2 -21867.153} C_VEL
LIN {X 0,Y 142.172,Z 747.949,A -85,B 0,C 180,E1 -21861.475,E2 -21861.475} C_VEL
LIN {X 0,Y 143.964,Z 745.061,A -85,B 0,C 180,E1 -21855.876,E2 -21855.876} C_VEL
LIN {X 0,Y 146.057,Z 741.828,A -85,B 0,C 180,E1 -21851.778,E2 -21851.778} C_VEL
LIN {X 0,Y 148.92,Z 737.622,A -85,B 0,C 180,E1 -21847.822,E2 -21847.822} C_VEL
LIN {X 0,Y 152.34,Z 732.342,A -85,B 0,C 180,E1 -21844.011,E2 -21844.011} C_VEL
LIN {X 0,Y 156.218,Z 725.825,A -85,B 0,C 180,E1 -21840.343,E2 -21840.343} C_VEL
LIN {X 0,Y 160.776,Z 717.812,A -85,B 0,C 180,E1 -21836.883,E2 -21836.883} C_VEL
LIN {X 0,Y 164.779,Z 709.809,A -85,B 0,C 180,E1 -21834.133,E2 -21834.133} C_VEL
LIN {X 0,Y 169.257,Z 699.966,A -85,B 0,C 180,E1 -21831.481,E2 -21831.481} C_VEL
LIN {X 0,Y 173.603,Z 689.198,A -85,B 0,C 180,E1 -21829.252,E2 -21829.252} C_VEL
LIN {X 0,Y 177.132,Z 678.847,A -85,B 0,C 180,E1 -21827.589,E2 -21827.589} C_VEL
LIN {X 0,Y 180.469,Z 666.719,A -85,B 0,C 180,E1 -21826.083,E2 -21826.083} C_VEL
LIN {X 0,Y 183.136,Z 653.493,A -85,B 0,C 180,E1 -21824.871,E2 -21824.871} C_VEL
LIN {X 0,Y 185.071,Z 639.462,A -85,B 0,C 180,E1 -21824.021,E2 -21824.021} C_VEL
LIN {X 0,Y 188.659,Z 589.153,A -85,B 0,C 180,E1 -21822.4,E2 -21822.4} C_VEL
LIN {X 0,Y 189.037,Z 582.867,A -85,B 0,C 180,E1 -21822.185,E2 -21822.185} C_VEL
LIN {X 0,Y 183.711,Z 570.429,A -85,B 0,C 180,E1 -21819.465,E2 -21819.465} C_VEL
LIN {X 0,Y 178.364,Z 559.983,A -85,B 0,C 180,E1 -21816.508,E2 -21816.508} C_VEL
LIN {X 0,Y 173.34,Z 551.261,A -85,B 0,C 180,E1 -21813.406,E2 -21813.406} C_VEL
LIN {X 0,Y 170.005,Z 546.013,A -85,B 0,C 180,E1 -21811.115,E2 -21811.115} C_VEL
LIN {X 0,Y 167.358,Z 541.963,A -85,B 0,C 180,E1 -21809.112,E2 -21809.112} C_VEL
LIN {X 0,Y 163.792,Z 536.821,A -85,B 0,C 180,E1 -21806.092,E2 -21806.092} C_VEL
LIN {X 0,Y 159.702,Z 531.411,A -85,B 0,C 180,E1 -21801.967,E2 -21801.967} C_VEL
LIN {X 0,Y 155.155,Z 525.575,A -85,B 0,C 180,E1 -21795.771,E2 -21795.771} C_VEL
LIN {X 0,Y 151.912,Z 522.058,A -85,B 0,C 180,E1 -21788.313,E2 -21788.313} C_VEL
LIN {X 0,Y 151.079,Z 520.498,A -85,B 0,C 180,E1 -21781.333,E2 -21781.333} C_VEL
LIN {X 0,Y 151.195,Z 520.535,A -85,B 0,C 180,E1 -21779.335,E2 -21779.335} C_VEL
LIN {X 0,Y 153.413,Z 523.881,A -85,B 0,C 180,E1 -21770.775,E2 -21770.775} C_VEL
LIN {X 0,Y 155.956,Z 526.818,A -85,B 0,C 180,E1 -21766.149,E2 -21766.149} C_VEL
LIN {X 0,Y 161.041,Z 533.523,A -85,B 0,C 180,E1 -21759.776,E2 -21759.776} C_VEL
LIN {X 0,Y 165.302,Z 539.383,A -85,B 0,C 180,E1 -21755.761,E2 -21755.761} C_VEL
LIN {X 0,Y 169.366,Z 545.636,A -85,B 0,C 180,E1 -21752.507,E2 -21752.507} C_VEL
LIN {X 0,Y 172.508,Z 550.618,A -85,B 0,C 180,E1 -21750.284,E2 -21750.284} C_VEL
LIN {X 0,Y 175.754,Z 556.157,A -85,B 0,C 180,E1 -21748.175,E2 -21748.175} C_VEL
LIN {X 0,Y 181.124,Z 566.13,A -85,B 0,C 180,E1 -21745.009,E2 -21745.009} C_VEL
LIN {X 0,Y 186.038,Z 576.829,A -85,B 0,C 180,E1 -21742.355,E2 -21742.355} C_VEL
LIN {X 0,Y 189.294,Z 584.788,A -85,B 0,C 180,E1 -21740.693,E2 -21740.693} C_VEL
LIN {X 0,Y 184.504,Z 647.709,A -85,B 0,C 180,E1 -21738.579,E2 -21738.579} C_VEL
LIN {X 0,Y 182.402,Z 661.928,A -85,B 0,C 180,E1 -21737.769,E2 -21737.769} C_VEL
LIN {X 0,Y 179.405,Z 675.52,A -85,B 0,C 180,E1 -21736.644,E2 -21736.644} C_VEL
LIN {X 0,Y 175.79,Z 688.154,A -85,B 0,C 180,E1 -21735.201,E2 -21735.201} C_VEL
LIN {X 0,Y 171.527,Z 700.381,A -85,B 0,C 180,E1 -21733.333,E2 -21733.333} C_VEL
LIN {X 0,Y 166.9,Z 711.79,A -85,B 0,C 180,E1 -21731.019,E2 -21731.019} C_VEL
LIN {X 0,Y 161.957,Z 722.68,A -85,B 0,C 180,E1 -21728.126,E2 -21728.126} C_VEL
LIN {X 0,Y 157.053,Z 732.406,A -85,B 0,C 180,E1 -21724.784,E2 -21724.784} C_VEL
LIN {X 0,Y 152.602,Z 740.519,A -85,B 0,C 180,E1 -21721.201,E2 -21721.201} C_VEL
LIN {X 0,Y 148.357,Z 748.226,A -85,B 0,C 180,E1 -21716.742,E2 -21716.742} C_VEL
LIN {X 0,Y 145.34,Z 753.516,A -85,B 0,C 180,E1 -21712.754,E2 -21712.754} C_VEL
LIN {X 0,Y 143.236,Z 757.767,A -85,B 0,C 180,E1 -21708.594,E2 -21708.594} C_VEL
LIN {X 0,Y 141.722,Z 761.076,A -85,B 0,C 180,E1 -21704.352,E2 -21704.352} C_VEL
LIN {X 0,Y 140.816,Z 764.118,A -85,B 0,C 180,E1 -21698.607,E2 -21698.607} C_VEL
LIN {X 0,Y 140.868,Z 765.505,A -85,B 0,C 180,E1 -21693.79,E2 -21693.79} C_VEL
LIN {X 0,Y 141.062,Z 765.887,A -85,B 0,C 180,E1 -21689.996,E2 -21689.996} C_VEL
LIN {X 0,Y 140.872,Z 765.514,A -85,B 0,C 180,E1 -21686.181,E2 -21686.181} C_VEL
LIN {X 0,Y 141.106,Z 764.165,A -85,B 0,C 180,E1 -21681.403,E2 -21681.403} C_VEL
LIN {X 0,Y 142.561,Z 761.175,A -85,B 0,C 180,E1 -21675.726,E2 -21675.726} C_VEL
LIN {X 0,Y 143.975,Z 759,A -85,B 0,C 180,E1 -21672.783,E2 -21672.783} C_VEL
LIN {X 0,Y 146.708,Z 761.634,A -85,B 0,C 180,E1 -21667.462,E2 -21667.462} C_VEL
LIN {X 0,Y 151.997,Z 763.348,A -85,B 0,C 180,E1 -21661.464,E2 -21661.464} C_VEL
LIN {X 0,Y 157.153,Z 763.696,A -85,B 0,C 180,E1 -21657.541,E2 -21657.541} C_VEL
LIN {X 0,Y 164.442,Z 763.093,A -85,B 0,C 180,E1 -21653.245,E2 -21653.245} C_VEL
LIN {X 0,Y 173.076,Z 761.408,A -85,B 0,C 180,E1 -21649.477,E2 -21649.477} C_VEL
LIN {X 0,Y 182.764,Z 758.603,A -85,B 0,C 180,E1 -21646.194,E2 -21646.194} C_VEL
LIN {X 0,Y 193.439,Z 754.58,A -85,B 0,C 180,E1 -21643.391,E2 -21643.391} C_VEL
LIN {X 0,Y 194.086,Z 754.242,A -85,B 0,C 180,E1 -21642.889,E2 -21642.889} C_VEL
LIN {X 0,Y 184.715,Z 757.01,A -85,B 0,C 180,E1 -21640.301,E2 -21640.301} C_VEL
LIN {X 0,Y 175.071,Z 758.822,A -85,B 0,C 180,E1 -21637.024,E2 -21637.024} C_VEL
LIN {X 0,Y 166.376,Z 759.311,A -85,B 0,C 180,E1 -21633.308,E2 -21633.308} C_VEL
LIN {X 0,Y 158.792,Z 758.521,A -85,B 0,C 180,E1 -21629.134,E2 -21629.134} C_VEL
LIN {X 0,Y 152.566,Z 756.466,A -85,B 0,C 180,E1 -21624.493,E2 -21624.493} C_VEL
LIN {X 0,Y 147.779,Z 753.147,A -85,B 0,C 180,E1 -21619.445,E2 -21619.445} C_VEL
LIN {X 0,Y 146.3,Z 751.422,A -85,B 0,C 180,E1 -21617.336,E2 -21617.336} C_VEL
LIN {X 0,Y 144.435,Z 749.426,A -85,B 0,C 180,E1 -21615.278,E2 -21615.278} C_VEL
LIN {X 0,Y 140.182,Z 745.305,A -85,B 0,C 180,E1 -21612.085,E2 -21612.085} C_VEL
LIN {X 0,Y 136.484,Z 740.458,A -85,B 0,C 180,E1 -21608.821,E2 -21608.821} C_VEL
LIN {X 0,Y 135.567,Z 737.395,A -85,B 0,C 180,E1 -21606.707,E2 -21606.707} C_VEL
LIN {X 0,Y 135.336,Z 730.591,A -85,B 0,C 180,E1 -21602.232,E2 -21602.232} C_VEL
LIN {X 0,Y 135.48,Z 723.721,A -85,B 0,C 180,E1 -21598.513,E2 -21598.513} C_VEL
LIN {X 0,Y 135.847,Z 713.754,A -85,B 0,C 180,E1 -21594.061,E2 -21594.061} C_VEL
LIN {X 0,Y 136.415,Z 704.322,A -85,B 0,C 180,E1 -21590.627,E2 -21590.627} C_VEL
LIN {X 0,Y 137.426,Z 690.843,A -85,B 0,C 180,E1 -21586.693,E2 -21586.693} C_VEL
LIN {X 0,Y 138.439,Z 678.109,A -85,B 0,C 180,E1 -21583.786,E2 -21583.786} C_VEL
LIN {X 0,Y 139.548,Z 663.907,A -85,B 0,C 180,E1 -21581.272,E2 -21581.272} C_VEL
LIN {X 0,Y 140.078,Z 656.483,A -85,B 0,C 180,E1 -21580.204,E2 -21580.204} C_VEL
LIN {X 0,Y 140.025,Z 657.976,A -85,B 0,C 180,E1 -21579.718,E2 -21579.718} C_VEL
LIN {X 0,Y 140.144,Z 658.309,A -85,B 0,C 180,E1 -21579.449,E2 -21579.449} C_VEL
LIN {X 0,Y 140.991,Z 657.857,A -85,B 0,C 180,E1 -21578.622,E2 -21578.622} C_VEL
LIN {X 0,Y 142.278,Z 656.133,A -85,B 0,C 180,E1 -21577.778,E2 -21577.778} C_VEL
LIN {X 0,Y 144.617,Z 651.641,A -85,B 0,C 180,E1 -21576.726,E2 -21576.726} C_VEL
LIN {X 0,Y 147.58,Z 643.537,A -85,B 0,C 180,E1 -21575.733,E2 -21575.733} C_VEL
LIN {X 0,Y 149.236,Z 637.972,A -85,B 0,C 180,E1 -21575.165,E2 -21575.165} C_VEL
LIN {X 0,Y 150.782,Z 636.101,A -85,B 0,C 180,E1 -21574.089,E2 -21574.089} C_VEL
LIN {X 0,Y 152.237,Z 633.241,A -85,B 0,C 180,E1 -21573.249,E2 -21573.249} C_VEL
LIN {X 0,Y 154.508,Z 626.968,A -85,B 0,C 180,E1 -21572.146,E2 -21572.146} C_VEL
LIN {X 0,Y 158.177,Z 614.345,A -85,B 0,C 180,E1 -21570.741,E2 -21570.741} C_VEL
LIN {X 0,Y 161.154,Z 602.856,A -85,B 0,C 180,E1 -21569.803,E2 -21569.803} C_VEL
LIN {X 0,Y 163.641,Z 598.965,A -85,B 0,C 180,E1 -21568.582,E2 -21568.582} C_VEL
LIN {X 0,Y 166.633,Z 591.938,A -85,B 0,C 180,E1 -21567.397,E2 -21567.397} C_VEL
LIN {X 0,Y 170.315,Z 580.769,A -85,B 0,C 180,E1 -21566.235,E2 -21566.235} C_VEL
LIN {X 0,Y 171.894,Z 575.563,A -85,B 0,C 180,E1 -21565.793,E2 -21565.793} C_VEL
LIN {X 0,Y 175.007,Z 570.907,A -85,B 0,C 180,E1 -21564.564,E2 -21564.564} C_VEL
LIN {X 0,Y 176.535,Z 567.89,A -85,B 0,C 180,E1 -21564.04,E2 -21564.04} C_VEL
LIN {X 0,Y 180.825,Z 576.714,A -85,B 0,C 180,E1 -21561.547,E2 -21561.547} C_VEL
LIN {X 0,Y 184.541,Z 585.672,A -85,B 0,C 180,E1 -21559.51,E2 -21559.51} C_VEL
LIN {X 0,Y 180.657,Z 639.136,A -85,B 0,C 180,E1 -21557.77,E2 -21557.77} C_VEL
LIN {X 0,Y 178.692,Z 652.641,A -85,B 0,C 180,E1 -21556.999,E2 -21556.999} C_VEL
LIN {X 0,Y 175.907,Z 666.166,A -85,B 0,C 180,E1 -21555.783,E2 -21555.783} C_VEL
LIN {X 0,Y 172.391,Z 678.529,A -85,B 0,C 180,E1 -21554.282,E2 -21554.282} C_VEL
LIN {X 0,Y 168.223,Z 690.294,A -85,B 0,C 180,E1 -21552.355,E2 -21552.355} C_VEL
LIN {X 0,Y 163.665,Z 700.937,A -85,B 0,C 180,E1 -21550.104,E2 -21550.104} C_VEL
LIN {X 0,Y 159.276,Z 710.22,A -85,B 0,C 180,E1 -21547.525,E2 -21547.525} C_VEL
LIN {X 0,Y 154.852,Z 718.594,A -85,B 0,C 180,E1 -21544.567,E2 -21544.567} C_VEL
LIN {X 0,Y 150.043,Z 726.541,A -85,B 0,C 180,E1 -21541.017,E2 -21541.017} C_VEL
LIN {X 0,Y 145.849,Z 733.006,A -85,B 0,C 180,E1 -21537.247,E2 -21537.247} C_VEL
LIN {X 0,Y 142.325,Z 738.23,A -85,B 0,C 180,E1 -21533.272,E2 -21533.272} C_VEL
LIN {X 0,Y 139.343,Z 742.385,A -85,B 0,C 180,E1 -21529.141,E2 -21529.141} C_VEL
LIN {X 0,Y 137.106,Z 745.571,A -85,B 0,C 180,E1 -21524.854,E2 -21524.854} C_VEL
LIN {X 0,Y 135.189,Z 748.42,A -85,B 0,C 180,E1 -21518.976,E2 -21518.976} C_VEL
LIN {X 0,Y 134.225,Z 749.836,A -85,B 0,C 180,E1 -21513.005,E2 -21513.005} C_VEL
LIN {X 0,Y 134.226,Z 749.808,A -85,B 0,C 180,E1 -21507.003,E2 -21507.003} C_VEL
LIN {X 0,Y 135.186,Z 748.357,A -85,B 0,C 180,E1 -21501.031,E2 -21501.031} C_VEL
LIN {X 0,Y 137.1,Z 745.471,A -85,B 0,C 180,E1 -21495.153,E2 -21495.153} C_VEL
LIN {X 0,Y 139.348,Z 742.238,A -85,B 0,C 180,E1 -21490.867,E2 -21490.867} C_VEL
LIN {X 0,Y 142.381,Z 738.035,A -85,B 0,C 180,E1 -21486.745,E2 -21486.745} C_VEL
LIN {X 0,Y 146,Z 732.759,A -85,B 0,C 180,E1 -21482.791,E2 -21482.791} C_VEL
LIN {X 0,Y 150.119,Z 726.247,A -85,B 0,C 180,E1 -21479.009,E2 -21479.009} C_VEL
LIN {X 0,Y 154.903,Z 718.243,A -85,B 0,C 180,E1 -21475.454,E2 -21475.454} C_VEL
LIN {X 0,Y 159.436,Z 709.574,A -85,B 0,C 180,E1 -21472.425,E2 -21472.425} C_VEL
LIN {X 0,Y 164.296,Z 699.367,A -85,B 0,C 180,E1 -21469.689,E2 -21469.689} C_VEL
LIN {X 0,Y 168.321,Z 689.685,A -85,B 0,C 180,E1 -21467.684,E2 -21467.684} C_VEL
LIN {X 0,Y 172.536,Z 677.7,A -85,B 0,C 180,E1 -21465.773,E2 -21465.773} C_VEL
LIN {X 0,Y 175.731,Z 666.217,A -85,B 0,C 180,E1 -21464.372,E2 -21464.372} C_VEL
LIN {X 0,Y 178.359,Z 653.484,A -85,B 0,C 180,E1 -21463.205,E2 -21463.205} C_VEL
LIN {X 0,Y 180.241,Z 640.483,A -85,B 0,C 180,E1 -21462.408,E2 -21462.408} C_VEL
LIN {X 0,Y 182.359,Z 613.652,A -85,B 0,C 180,E1 -21461.499,E2 -21461.499} C_VEL
LIN {X 0,Y 184.297,Z 585.28,A -85,B 0,C 180,E1 -21460.581,E2 -21460.581} C_VEL
LIN {X 0,Y 179.737,Z 574.461,A -85,B 0,C 180,E1 -21458.066,E2 -21458.066} C_VEL
LIN {X 0,Y 174.677,Z 564.338,A -85,B 0,C 180,E1 -21455.046,E2 -21455.046} C_VEL
LIN {X 0,Y 170.162,Z 556.287,A -85,B 0,C 180,E1 -21452.038,E2 -21452.038} C_VEL
LIN {X 0,Y 167.2,Z 551.434,A -85,B 0,C 180,E1 -21449.848,E2 -21449.848} C_VEL
LIN {X 0,Y 164.784,Z 547.692,A -85,B 0,C 180,E1 -21447.89,E2 -21447.89} C_VEL
LIN {X 0,Y 161.535,Z 542.805,A -85,B 0,C 180,E1 -21444.929,E2 -21444.929} C_VEL
LIN {X 0,Y 158.06,Z 537.978,A -85,B 0,C 180,E1 -21441.179,E2 -21441.179} C_VEL
LIN {X 0,Y 153.929,Z 532.416,A -85,B 0,C 180,E1 -21435.221,E2 -21435.221} C_VEL
LIN {X 0,Y 150.806,Z 528.764,A -85,B 0,C 180,E1 -21427.341,E2 -21427.341} C_VEL
LIN {X 0,Y 150.287,Z 527.435,A -85,B 0,C 180,E1 -21420,E2 -21420} C_VEL
LIN {X 0,Y 152.414,Z 530.907,A -85,B 0,C 180,E1 -21411.005,E2 -21411.005} C_VEL
LIN {X 0,Y 154.671,Z 533.683,A -85,B 0,C 180,E1 -21406.701,E2 -21406.701} C_VEL
LIN {X 0,Y 159.272,Z 540.015,A -85,B 0,C 180,E1 -21400.6,E2 -21400.6} C_VEL
LIN {X 0,Y 163.331,Z 545.92,A -85,B 0,C 180,E1 -21396.546,E2 -21396.546} C_VEL
LIN {X 0,Y 167.195,Z 552.06,A -85,B 0,C 180,E1 -21393.29,E2 -21393.29} C_VEL
LIN {X 0,Y 170.85,Z 558.172,A -85,B 0,C 180,E1 -21390.59,E2 -21390.59} C_VEL
LIN {X 0,Y 175.348,Z 566.514,A -85,B 0,C 180,E1 -21387.61,E2 -21387.61} C_VEL
LIN {X 0,Y 179.533,Z 575.175,A -85,B 0,C 180,E1 -21385.083,E2 -21385.083} C_VEL
LIN {X 0,Y 183.846,Z 585.461,A -85,B 0,C 180,E1 -21382.656,E2 -21382.656} C_VEL
LIN {X 0,Y 184.528,Z 587.232,A -85,B 0,C 180,E1 -21382.284,E2 -21382.284} C_VEL
LIN {X 0,Y 179.719,Z 647.832,A -85,B 0,C 180,E1 -21380.229,E2 -21380.229} C_VEL
LIN {X 0,Y 177.54,Z 661.931,A -85,B 0,C 180,E1 -21379.419,E2 -21379.419} C_VEL
LIN {X 0,Y 174.31,Z 676.022,A -85,B 0,C 180,E1 -21378.231,E2 -21378.231} C_VEL
LIN {X 0,Y 170.287,Z 689.328,A -85,B 0,C 180,E1 -21376.665,E2 -21376.665} C_VEL
LIN {X 0,Y 165.887,Z 701.2,A -85,B 0,C 180,E1 -21374.771,E2 -21374.771} C_VEL
LIN {X 0,Y 161.235,Z 712.08,A -85,B 0,C 180,E1 -21372.497,E2 -21372.497} C_VEL
LIN {X 0,Y 156.311,Z 722.419,A -85,B 0,C 180,E1 -21369.682,E2 -21369.682} C_VEL
LIN {X 0,Y 151.223,Z 731.967,A -85,B 0,C 180,E1 -21366.333,E2 -21366.333} C_VEL
LIN {X 0,Y 146.52,Z 740.089,A -85,B 0,C 180,E1 -21362.653,E2 -21362.653} C_VEL
LIN {X 0,Y 141.998,Z 747.805,A -85,B 0,C 180,E1 -21358.042,E2 -21358.042} C_VEL
LIN {X 0,Y 138.757,Z 753.096,A -85,B 0,C 180,E1 -21353.899,E2 -21353.899} C_VEL
LIN {X 0,Y 136.456,Z 757.35,A -85,B 0,C 180,E1 -21349.555,E2 -21349.555} C_VEL
LIN {X 0,Y 134.792,Z 760.661,A -85,B 0,C 180,E1 -21345.107,E2 -21345.107} C_VEL
LIN {X 0,Y 133.772,Z 763.706,A -85,B 0,C 180,E1 -21339.064,E2 -21339.064} C_VEL
LIN {X 0,Y 133.784,Z 765.262,A -85,B 0,C 180,E1 -21333.007,E2 -21333.007} C_VEL
LIN {X 0,Y 133.981,Z 765.478,A -85,B 0,C 180,E1 -21329.996,E2 -21329.996} C_VEL
LIN {X 0,Y 133.809,Z 765.162,A -85,B 0,C 180,E1 -21326.308,E2 -21326.308} C_VEL
LIN {X 0,Y 134.078,Z 763.755,A -85,B 0,C 180,E1 -21320.949,E2 -21320.949} C_VEL
LIN {X 0,Y 135.678,Z 760.764,A -85,B 0,C 180,E1 -21314.986,E2 -21314.986} C_VEL
LIN {X 0,Y 137.874,Z 757.801,A -85,B 0,C 180,E1 -21310.84,E2 -21310.84} C_VEL
LIN {X 0,Y 140.322,Z 760.128,A -85,B 0,C 180,E1 -21306.376,E2 -21306.376} C_VEL
LIN {X 0,Y 144.943,Z 762.088,A -85,B 0,C 180,E1 -21300.992,E2 -21300.992} C_VEL
LIN {X 0,Y 151.237,Z 763.003,A -85,B 0,C 180,E1 -21296.103,E2 -21296.103} C_VEL
LIN {X 0,Y 158.811,Z 762.861,A -85,B 0,C 180,E1 -21291.713,E2 -21291.713} C_VEL
LIN {X 0,Y 167.759,Z 761.673,A -85,B 0,C 180,E1 -21287.906,E2 -21287.906} C_VEL
LIN {X 0,Y 177.733,Z 759.412,A -85,B 0,C 180,E1 -21284.618,E2 -21284.618} C_VEL
LIN {X 0,Y 183.128,Z 757.859,A -85,B 0,C 180,E1 -21283.179,E2 -21283.179} C_VEL
LIN {X 0,Y 179.442,Z 758.511,A -85,B 0,C 180,E1 -21281.745,E2 -21281.745} C_VEL
LIN {X 0,Y 169.51,Z 759.77,A -85,B 0,C 180,E1 -21278.455,E2 -21278.455} C_VEL
LIN {X 0,Y 160.508,Z 759.747,A -85,B 0,C 180,E1 -21274.695,E2 -21274.695} C_VEL
LIN {X 0,Y 152.639,Z 758.457,A -85,B 0,C 180,E1 -21270.429,E2 -21270.429} C_VEL
LIN {X 0,Y 146.159,Z 755.944,A -85,B 0,C 180,E1 -21265.643,E2 -21265.643} C_VEL
LIN {X 0,Y 141.181,Z 752.164,A -85,B 0,C 180,E1 -21260.393,E2 -21260.393} C_VEL
LIN {X 0,Y 137.783,Z 747.044,A -85,B 0,C 180,E1 -21254.775,E2 -21254.775} C_VEL
LIN {X 0,Y 135.811,Z 740.323,A -85,B 0,C 180,E1 -21248.931,E2 -21248.931} C_VEL
LIN {X 0,Y 135.567,Z 737.395,A -85,B 0,C 180,E1 -21246.707,E2 -21246.707} C_VEL
LIN {X 0,Y 135.177,Z 735.328,A -85,B 0,C 180,E1 -21245.313,E2 -21245.313} C_VEL
LIN {X 0,Y 133.814,Z 731.822,A -85,B 0,C 180,E1 -21243.364,E2 -21243.364} C_VEL
LIN {X 0,Y 129.733,Z 722.544,A -85,B 0,C 180,E1 -21239.131,E2 -21239.131} C_VEL
LIN {X 0,Y 128.87,Z 718.289,A -85,B 0,C 180,E1 -21237.283,E2 -21237.283} C_VEL
LIN {X 0,Y 128.857,Z 716.864,A -85,B 0,C 180,E1 -21236.654,E2 -21236.654} C_VEL
LIN {X 0,Y 129.425,Z 705.842,A -85,B 0,C 180,E1 -21232.197,E2 -21232.197} C_VEL
LIN {X 0,Y 130.129,Z 694.151,A -85,B 0,C 180,E1 -21228.41,E2 -21228.41} C_VEL
LIN {X 0,Y 131.135,Z 681.889,A -85,B 0,C 180,E1 -21225.221,E2 -21225.221} C_VEL
LIN {X 0,Y 131.755,Z 672.952,A -85,B 0,C 180,E1 -21223.27,E2 -21223.27} C_VEL
LIN {X 0,Y 131.682,Z 673.565,A -85,B 0,C 180,E1 -21222.931,E2 -21222.931} C_VEL
LIN {X 0,Y 132.552,Z 673.771,A -85,B 0,C 180,E1 -21221.45,E2 -21221.45} C_VEL
LIN {X 0,Y 133.471,Z 672.88,A -85,B 0,C 180,E1 -21220.729,E2 -21220.729} C_VEL
LIN {X 0,Y 135.729,Z 669.952,A -85,B 0,C 180,E1 -21219.486,E2 -21219.486} C_VEL
LIN {X 0,Y 138.511,Z 665.345,A -85,B 0,C 180,E1 -21218.416,E2 -21218.416} C_VEL
LIN {X 0,Y 141.139,Z 662.992,A -85,B 0,C 180,E1 -21216.524,E2 -21216.524} C_VEL
LIN {X 0,Y 143.456,Z 659.87,A -85,B 0,C 180,E1 -21215.36,E2 -21215.36} C_VEL
LIN {X 0,Y 146.312,Z 654.711,A -85,B 0,C 180,E1 -21214.293,E2 -21214.293} C_VEL
LIN {X 0,Y 149.816,Z 646.067,A -85,B 0,C 180,E1 -21213.334,E2 -21213.334} C_VEL
LIN {X 0,Y 150.884,Z 642.92,A -85,B 0,C 180,E1 -21213.01,E2 -21213.01} C_VEL
LIN {X 0,Y 153.444,Z 639.139,A -85,B 0,C 180,E1 -21211.628,E2 -21211.628} C_VEL
LIN {X 0,Y 156.129,Z 632.953,A -85,B 0,C 180,E1 -21210.412,E2 -21210.412} C_VEL
LIN {X 0,Y 159.728,Z 621.778,A -85,B 0,C 180,E1 -21209.052,E2 -21209.052} C_VEL
LIN {X 0,Y 163.773,Z 607.033,A -85,B 0,C 180,E1 -21207.832,E2 -21207.832} C_VEL
LIN {X 0,Y 166.665,Z 602.109,A -85,B 0,C 180,E1 -21206.576,E2 -21206.576} C_VEL
LIN {X 0,Y 170.22,Z 593.69,A -85,B 0,C 180,E1 -21205.319,E2 -21205.319} C_VEL
LIN {X 0,Y 174.033,Z 582.162,A -85,B 0,C 180,E1 -21204.246,E2 -21204.246} C_VEL
LIN {X 0,Y 174.9,Z 579.621,A -85,B 0,C 180,E1 -21204.007,E2 -21204.007} C_VEL
LIN {X 0,Y 175.475,Z 578.828,A -85,B 0,C 180,E1 -21203.789,E2 -21203.789} C_VEL
LIN {X 0,Y 175.996,Z 578.636,A -85,B 0,C 180,E1 -21203.558,E2 -21203.558} C_VEL
LIN {X 0,Y 179.604,Z 587.259,A -85,B 0,C 180,E1 -21201.399,E2 -21201.399} C_VEL
LIN {X 0,Y 179.964,Z 588.171,A -85,B 0,C 180,E1 -21201.192,E2 -21201.192} C_VEL
LIN {X 0,Y 176.097,Z 639.25,A -85,B 0,C 180,E1 -21199.514,E2 -21199.514} C_VEL
LIN {X 0,Y 174.097,Z 652.614,A -85,B 0,C 180,E1 -21198.755,E2 -21198.755} C_VEL
LIN {X 0,Y 171.338,Z 665.65,A -85,B 0,C 180,E1 -21197.593,E2 -21197.593} C_VEL
LIN {X 0,Y 167.974,Z 677.319,A -85,B 0,C 180,E1 -21196.202,E2 -21196.202} C_VEL
LIN {X 0,Y 163.63,Z 689.479,A -85,B 0,C 180,E1 -21194.267,E2 -21194.267} C_VEL
LIN {X 0,Y 158.845,Z 700.332,A -85,B 0,C 180,E1 -21192.009,E2 -21192.009} C_VEL
LIN {X 0,Y 154.445,Z 709.274,A -85,B 0,C 180,E1 -21189.577,E2 -21189.577} C_VEL
LIN {X 0,Y 149.086,Z 719.02,A -85,B 0,C 180,E1 -21186.108,E2 -21186.108} C_VEL
LIN {X 0,Y 144.022,Z 726.96,A -85,B 0,C 180,E1 -21182.469,E2 -21182.469} C_VEL
LIN {X 0,Y 139.589,Z 733.421,A -85,B 0,C 180,E1 -21178.579,E2 -21178.579} C_VEL
LIN {X 0,Y 135.828,Z 738.643,A -85,B 0,C 180,E1 -21174.456,E2 -21174.456} C_VEL
LIN {X 0,Y 132.679,Z 742.794,A -85,B 0,C 180,E1 -21170.143,E2 -21170.143} C_VEL
LIN {X 0,Y 130.253,Z 745.981,A -85,B 0,C 180,E1 -21165.655,E2 -21165.655} C_VEL
LIN {X 0,Y 128.192,Z 748.829,A -85,B 0,C 180,E1 -21159.471,E2 -21159.471} C_VEL
LIN {X 0,Y 127.161,Z 750.244,A -85,B 0,C 180,E1 -21153.172,E2 -21153.172} C_VEL
LIN {X 0,Y 127.162,Z 750.217,A -85,B 0,C 180,E1 -21146.836,E2 -21146.836} C_VEL
LIN {X 0,Y 128.189,Z 748.767,A -85,B 0,C 180,E1 -21140.537,E2 -21140.537} C_VEL
LIN {X 0,Y 130.246,Z 745.881,A -85,B 0,C 180,E1 -21134.352,E2 -21134.352} C_VEL
LIN {X 0,Y 132.685,Z 742.649,A -85,B 0,C 180,E1 -21129.866,E2 -21129.866} C_VEL
LIN {X 0,Y 135.903,Z 738.449,A -85,B 0,C 180,E1 -21125.567,E2 -21125.567} C_VEL
LIN {X 0,Y 139.709,Z 733.18,A -85,B 0,C 180,E1 -21121.457,E2 -21121.457} C_VEL
LIN {X 0,Y 144.096,Z 726.671,A -85,B 0,C 180,E1 -21117.559,E2 -21117.559} C_VEL
LIN {X 0,Y 149.134,Z 718.674,A -85,B 0,C 180,E1 -21113.914,E2 -21113.914} C_VEL
LIN {X 0,Y 153.816,Z 710.138,A -85,B 0,C 180,E1 -21110.854,E2 -21110.854} C_VEL
LIN {X 0,Y 158.425,Z 700.89,A -85,B 0,C 180,E1 -21108.29,E2 -21108.29} C_VEL
LIN {X 0,Y 163.161,Z 690.173,A -85,B 0,C 180,E1 -21106.012,E2 -21106.012} C_VEL
LIN {X 0,Y 167.553,Z 678.252,A -85,B 0,C 180,E1 -21104.09,E2 -21104.09} C_VEL
LIN {X 0,Y 170.866,Z 666.844,A -85,B 0,C 180,E1 -21102.679,E2 -21102.679} C_VEL
LIN {X 0,Y 173.742,Z 653.475,A -85,B 0,C 180,E1 -21101.449,E2 -21101.449} C_VEL
LIN {X 0,Y 175.697,Z 640.345,A -85,B 0,C 180,E1 -21100.65,E2 -21100.65} C_VEL
LIN {X 0,Y 178.336,Z 607.657,A -85,B 0,C 180,E1 -21099.567,E2 -21099.567} C_VEL
LIN {X 0,Y 179.681,Z 587.7,A -85,B 0,C 180,E1 -21098.881,E2 -21098.881} C_VEL
LIN {X 0,Y 175.614,Z 577.897,A -85,B 0,C 180,E1 -21096.44,E2 -21096.44} C_VEL
LIN {X 0,Y 170.335,Z 567.119,A -85,B 0,C 180,E1 -21092.985,E2 -21092.985} C_VEL
LIN {X 0,Y 165.877,Z 559.041,A -85,B 0,C 180,E1 -21089.664,E2 -21089.664} C_VEL
LIN {X 0,Y 162.407,Z 553.52,A -85,B 0,C 180,E1 -21086.729,E2 -21086.729} C_VEL
LIN {X 0,Y 159.636,Z 549.182,A -85,B 0,C 180,E1 -21084.032,E2 -21084.032} C_VEL
LIN {X 0,Y 156.513,Z 544.634,A -85,B 0,C 180,E1 -21080.458,E2 -21080.458} C_VEL
LIN {X 0,Y 152.721,Z 539.237,A -85,B 0,C 180,E1 -21074.663,E2 -21074.663} C_VEL
LIN {X 0,Y 149.867,Z 535.748,A -85,B 0,C 180,E1 -21067.037,E2 -21067.037} C_VEL
LIN {X 0,Y 149.419,Z 534.505,A -85,B 0,C 180,E1 -21060,E2 -21060} C_VEL
LIN {X 0,Y 151.394,Z 537.891,A -85,B 0,C 180,E1 -21051.294,E2 -21051.294} C_VEL
LIN {X 0,Y 153.31,Z 540.4,A -85,B 0,C 180,E1 -21047.424,E2 -21047.424} C_VEL
LIN {X 0,Y 157.531,Z 546.505,A -85,B 0,C 180,E1 -21041.447,E2 -21041.447} C_VEL
LIN {X 0,Y 161.241,Z 552.189,A -85,B 0,C 180,E1 -21037.496,E2 -21037.496} C_VEL
LIN {X 0,Y 164.611,Z 557.757,A -85,B 0,C 180,E1 -21034.462,E2 -21034.462} C_VEL
LIN {X 0,Y 168.76,Z 564.972,A -85,B 0,C 180,E1 -21031.216,E2 -21031.216} C_VEL
LIN {X 0,Y 173.58,Z 574.6,A -85,B 0,C 180,E1 -21027.878,E2 -21027.878} C_VEL
LIN {X 0,Y 177.823,Z 584.261,A -85,B 0,C 180,E1 -21025.208,E2 -21025.208} C_VEL
LIN {X 0,Y 179.912,Z 589.648,A -85,B 0,C 180,E1 -21023.957,E2 -21023.957} C_VEL
LIN {X 0,Y 175.292,Z 646.246,A -85,B 0,C 180,E1 -21022.053,E2 -21022.053} C_VEL
LIN {X 0,Y 173.223,Z 660.069,A -85,B 0,C 180,E1 -21021.285,E2 -21021.285} C_VEL
LIN {X 0,Y 170.228,Z 673.128,A -85,B 0,C 180,E1 -21020.254,E2 -21020.254} C_VEL
LIN {X 0,Y 166.068,Z 687.042,A -85,B 0,C 180,E1 -21018.687,E2 -21018.687} C_VEL
LIN {X 0,Y 161.468,Z 699.376,A -85,B 0,C 180,E1 -21016.802,E2 -21016.802} C_VEL
LIN {X 0,Y 156.54,Z 710.529,A -85,B 0,C 180,E1 -21014.542,E2 -21014.542} C_VEL
LIN {X 0,Y 151.456,Z 720.924,A -85,B 0,C 180,E1 -21011.737,E2 -21011.737} C_VEL
LIN {X 0,Y 146.451,Z 730.022,A -85,B 0,C 180,E1 -21008.593,E2 -21008.593} C_VEL
LIN {X 0,Y 141.283,Z 738.4,A -85,B 0,C 180,E1 -21004.889,E2 -21004.889} C_VEL
LIN {X 0,Y 136.369,Z 746.363,A -85,B 0,C 180,E1 -21000.16,E2 -21000.16} C_VEL
LIN {X 0,Y 132.223,Z 752.675,A -85,B 0,C 180,E1 -20995.16,E2 -20995.16} C_VEL
LIN {X 0,Y 129.707,Z 756.932,A -85,B 0,C 180,E1 -20990.617,E2 -20990.617} C_VEL
LIN {X 0,Y 127.894,Z 760.246,A -85,B 0,C 180,E1 -20985.943,E2 -20985.943} C_VEL
LIN {X 0,Y 126.723,Z 763.293,A -85,B 0,C 180,E1 -20979.573,E2 -20979.573} C_VEL
LIN {X 0,Y 126.698,Z 764.852,A -85,B 0,C 180,E1 -20973.176,E2 -20973.176} C_VEL
LIN {X 0,Y 126.882,Z 765.069,A -85,B 0,C 180,E1 -20969.996,E2 -20969.996} C_VEL
LIN {X 0,Y 126.74,Z 764.817,A -85,B 0,C 180,E1 -20966.495,E2 -20966.495} C_VEL
LIN {X 0,Y 127.052,Z 763.344,A -85,B 0,C 180,E1 -20960.444,E2 -20960.444} C_VEL
LIN {X 0,Y 128.804,Z 760.353,A -85,B 0,C 180,E1 -20954.164,E2 -20954.164} C_VEL
LIN {X 0,Y 131.953,Z 756.514,A -85,B 0,C 180,E1 -20948.721,E2 -20948.721} C_VEL
LIN {X 0,Y 136.236,Z 759.721,A -85,B 0,C 180,E1 -20942.332,E2 -20942.332} C_VEL
LIN {X 0,Y 141.966,Z 761.555,A -85,B 0,C 180,E1 -20937.002,E2 -20937.002} C_VEL
LIN {X 0,Y 149.222,Z 762.377,A -85,B 0,C 180,E1 -20932.242,E2 -20932.242} C_VEL
LIN {X 0,Y 157.8,Z 762.195,A -85,B 0,C 180,E1 -20928.079,E2 -20928.079} C_VEL
LIN {X 0,Y 167.591,Z 760.991,A -85,B 0,C 180,E1 -20924.525,E2 -20924.525} C_VEL
LIN {X 0,Y 172.841,Z 760.004,A -85,B 0,C 180,E1 -20922.949,E2 -20922.949} C_VEL
LIN {X 0,Y 164.038,Z 760.498,A -85,B 0,C 180,E1 -20919.99,E2 -20919.99} C_VEL
LIN {X 0,Y 154.728,Z 759.966,A -85,B 0,C 180,E1 -20916.191,E2 -20916.191} C_VEL
LIN {X 0,Y 146.576,Z 758.189,A -85,B 0,C 180,E1 -20911.831,E2 -20911.831} C_VEL
LIN {X 0,Y 139.846,Z 755.198,A -85,B 0,C 180,E1 -20906.891,E2 -20906.891} C_VEL
LIN {X 0,Y 134.644,Z 750.971,A -85,B 0,C 180,E1 -20901.43,E2 -20901.43} C_VEL
LIN {X 0,Y 131.108,Z 745.431,A -85,B 0,C 180,E1 -20895.546,E2 -20895.546} C_VEL
LIN {X 0,Y 129.096,Z 738.26,A -85,B 0,C 180,E1 -20889.399,E2 -20889.399} C_VEL
LIN {X 0,Y 128.708,Z 731.705,A -85,B 0,C 180,E1 -20884.698,E2 -20884.698} C_VEL
LIN {X 0,Y 128.695,Z 723.71,A -85,B 0,C 180,E1 -20880,E2 -20880} C_VEL
LIN {X 0,Y 128.857,Z 716.864,A -85,B 0,C 180,E1 -20876.654,E2 -20876.654} C_VEL
LIN {X 0,Y 128.431,Z 712.569,A -85,B 0,C 180,E1 -20874.917,E2 -20874.917} C_VEL
LIN {X 0,Y 127.137,Z 707.96,A -85,B 0,C 180,E1 -20873.36,E2 -20873.36} C_VEL
LIN {X 0,Y 123.71,Z 696.432,A -85,B 0,C 180,E1 -20870.01,E2 -20870.01} C_VEL
LIN {X 0,Y 123.406,Z 691.305,A -85,B 0,C 180,E1 -20868.55,E2 -20868.55} C_VEL
LIN {X 0,Y 123.886,Z 685.043,A -85,B 0,C 180,E1 -20866.778,E2 -20866.778} C_VEL
LIN {X 0,Y 123.717,Z 685.924,A -85,B 0,C 180,E1 -20866.014,E2 -20866.014} C_VEL
LIN {X 0,Y 123.916,Z 686.059,A -85,B 0,C 180,E1 -20865.411,E2 -20865.411} C_VEL
LIN {X 0,Y 125.436,Z 684.888,A -85,B 0,C 180,E1 -20863.731,E2 -20863.731} C_VEL
LIN {X 0,Y 127.606,Z 682.471,A -85,B 0,C 180,E1 -20862.367,E2 -20862.367} C_VEL
LIN {X 0,Y 128.903,Z 680.771,A -85,B 0,C 180,E1 -20861.729,E2 -20861.729} C_VEL
LIN {X 0,Y 131.282,Z 679.184,A -85,B 0,C 180,E1 -20859.521,E2 -20859.521} C_VEL
LIN {X 0,Y 134.369,Z 676.069,A -85,B 0,C 180,E1 -20857.714,E2 -20857.714} C_VEL
LIN {X 0,Y 137.306,Z 672.09,A -85,B 0,C 180,E1 -20856.548,E2 -20856.548} C_VEL
LIN {X 0,Y 138.597,Z 670.325,A -85,B 0,C 180,E1 -20856.067,E2 -20856.067} C_VEL
LIN {X 0,Y 140.525,Z 668.714,A -85,B 0,C 180,E1 -20854.842,E2 -20854.842} C_VEL
LIN {X 0,Y 142.855,Z 666.109,A -85,B 0,C 180,E1 -20853.719,E2 -20853.719} C_VEL
LIN {X 0,Y 146.511,Z 660.792,A -85,B 0,C 180,E1 -20852.39,E2 -20852.39} C_VEL
LIN {X 0,Y 150.071,Z 653.859,A -85,B 0,C 180,E1 -20851.455,E2 -20851.455} C_VEL
LIN {X 0,Y 152.874,Z 647.099,A -85,B 0,C 180,E1 -20850.796,E2 -20850.796} C_VEL
LIN {X 0,Y 155.715,Z 642.841,A -85,B 0,C 180,E1 -20849.513,E2 -20849.513} C_VEL
LIN {X 0,Y 158.88,Z 636.035,A -85,B 0,C 180,E1 -20848.312,E2 -20848.312} C_VEL
LIN {X 0,Y 162.693,Z 624.723,A -85,B 0,C 180,E1 -20847.018,E2 -20847.018} C_VEL
LIN {X 0,Y 166.733,Z 610.794,A -85,B 0,C 180,E1 -20845.869,E2 -20845.869} C_VEL
LIN {X 0,Y 169.837,Z 605.257,A -85,B 0,C 180,E1 -20844.667,E2 -20844.667} C_VEL
LIN {X 0,Y 173.663,Z 596.322,A -85,B 0,C 180,E1 -20843.44,E2 -20843.44} C_VEL
LIN {X 0,Y 175.439,Z 591.33,A -85,B 0,C 180,E1 -20842.957,E2 -20842.957} C_VEL
LIN {X 0,Y 171.666,Z 639.699,A -85,B 0,C 180,E1 -20841.334,E2 -20841.334} C_VEL
LIN {X 0,Y 169.529,Z 653.347,A -85,B 0,C 180,E1 -20840.548,E2 -20840.548} C_VEL
LIN {X 0,Y 166.649,Z 666.263,A -85,B 0,C 180,E1 -20839.39,E2 -20839.39} C_VEL
LIN {X 0,Y 163.164,Z 677.86,A -85,B 0,C 180,E1 -20837.993,E2 -20837.993} C_VEL
LIN {X 0,Y 158.636,Z 689.965,A -85,B 0,C 180,E1 -20836.052,E2 -20836.052} C_VEL
LIN {X 0,Y 153.653,Z 700.788,A -85,B 0,C 180,E1 -20833.778,E2 -20833.778} C_VEL
LIN {X 0,Y 149.058,Z 709.712,A -85,B 0,C 180,E1 -20831.311,E2 -20831.311} C_VEL
LIN {X 0,Y 143.43,Z 719.447,A -85,B 0,C 180,E1 -20827.774,E2 -20827.774} C_VEL
LIN {X 0,Y 138.09,Z 727.38,A -85,B 0,C 180,E1 -20824.049,E2 -20824.049} C_VEL
LIN {X 0,Y 133.416,Z 733.834,A -85,B 0,C 180,E1 -20820.033,E2 -20820.033} C_VEL
LIN {X 0,Y 129.396,Z 739.055,A -85,B 0,C 180,E1 -20815.758,E2 -20815.758} C_VEL
LIN {X 0,Y 126.048,Z 743.203,A -85,B 0,C 180,E1 -20811.253,E2 -20811.253} C_VEL
LIN {X 0,Y 123.436,Z 746.389,A -85,B 0,C 180,E1 -20806.544,E2 -20806.544} C_VEL
LIN {X 0,Y 121.207,Z 749.238,A -85,B 0,C 180,E1 -20800.022,E2 -20800.022} C_VEL
LIN {X 0,Y 120.101,Z 750.652,A -85,B 0,C 180,E1 -20793.359,E2 -20793.359} C_VEL
LIN {X 0,Y 120.101,Z 750.625,A -85,B 0,C 180,E1 -20786.65,E2 -20786.65} C_VEL
LIN {X 0,Y 121.204,Z 749.176,A -85,B 0,C 180,E1 -20779.987,E2 -20779.987} C_VEL
LIN {X 0,Y 123.427,Z 746.292,A -85,B 0,C 180,E1 -20773.464,E2 -20773.464} C_VEL
LIN {X 0,Y 126.055,Z 743.061,A -85,B 0,C 180,E1 -20768.757,E2 -20768.757} C_VEL
LIN {X 0,Y 129.47,Z 738.865,A -85,B 0,C 180,E1 -20764.266,E2 -20764.266} C_VEL
LIN {X 0,Y 133.511,Z 733.599,A -85,B 0,C 180,E1 -20760,E2 -20760} C_VEL
LIN {X 0,Y 138.166,Z 727.096,A -85,B 0,C 180,E1 -20755.982,E2 -20755.982} C_VEL
LIN {X 0,Y 143.482,Z 719.106,A -85,B 0,C 180,E1 -20752.251,E2 -20752.251} C_VEL
LIN {X 0,Y 149.102,Z 709.305,A -85,B 0,C 180,E1 -20748.713,E2 -20748.713} C_VEL
LIN {X 0,Y 154.286,Z 699.188,A -85,B 0,C 180,E1 -20746.005,E2 -20746.005} C_VEL
LIN {X 0,Y 159.287,Z 687.919,A -85,B 0,C 180,E1 -20743.745,E2 -20743.745} C_VEL
LIN {X 0,Y 163.272,Z 677.047,A -85,B 0,C 180,E1 -20742.059,E2 -20742.059} C_VEL
LIN {X 0,Y 166.73,Z 665.216,A -85,B 0,C 180,E1 -20740.653,E2 -20740.653} C_VEL
LIN {X 0,Y 169.421,Z 652.706,A -85,B 0,C 180,E1 -20739.534,E2 -20739.534} C_VEL
LIN {X 0,Y 171.446,Z 639.3,A -85,B 0,C 180,E1 -20738.757,E2 -20738.757} C_VEL
LIN {X 0,Y 175.304,Z 590.414,A -85,B 0,C 180,E1 -20737.147,E2 -20737.147} C_VEL
LIN {X 0,Y 171.79,Z 581.732,A -85,B 0,C 180,E1 -20734.85,E2 -20734.85} C_VEL
LIN {X 0,Y 167.215,Z 572.118,A -85,B 0,C 180,E1 -20731.605,E2 -20731.605} C_VEL
LIN {X 0,Y 163.11,Z 564.415,A -85,B 0,C 180,E1 -20728.292,E2 -20728.292} C_VEL
LIN {X 0,Y 160.233,Z 559.614,A -85,B 0,C 180,E1 -20725.667,E2 -20725.667} C_VEL
LIN {X 0,Y 157.655,Z 555.357,A -85,B 0,C 180,E1 -20722.973,E2 -20722.973} C_VEL
LIN {X 0,Y 154.995,Z 551.274,A -85,B 0,C 180,E1 -20719.727,E2 -20719.727} C_VEL
LIN {X 0,Y 151.355,Z 545.911,A -85,B 0,C 180,E1 -20713.768,E2 -20713.768} C_VEL
LIN {X 0,Y 148.934,Z 542.753,A -85,B 0,C 180,E1 -20706.729,E2 -20706.729} C_VEL
LIN {X 0,Y 148.482,Z 541.653,A -85,B 0,C 180,E1 -20701.357,E2 -20701.357} C_VEL
LIN {X 0,Y 148.606,Z 541.932,A -85,B 0,C 180,E1 -20698.984,E2 -20698.984} C_VEL
LIN {X 0,Y 150.376,Z 544.894,A -85,B 0,C 180,E1 -20691.588,E2 -20691.588} C_VEL
LIN {X 0,Y 152.059,Z 547.26,A -85,B 0,C 180,E1 -20687.996,E2 -20687.996} C_VEL
LIN {X 0,Y 155.914,Z 553.159,A -85,B 0,C 180,E1 -20682.202,E2 -20682.202} C_VEL
LIN {X 0,Y 159.346,Z 558.668,A -85,B 0,C 180,E1 -20678.323,E2 -20678.323} C_VEL
LIN {X 0,Y 162.661,Z 564.472,A -85,B 0,C 180,E1 -20675.165,E2 -20675.165} C_VEL
LIN {X 0,Y 166.042,Z 570.711,A -85,B 0,C 180,E1 -20672.344,E2 -20672.344} C_VEL
LIN {X 0,Y 170.557,Z 580.126,A -85,B 0,C 180,E1 -20668.998,E2 -20668.998} C_VEL
